(* CoDeSys 2.3.9.62 project: P_auto.pro *)
(* Libraries: Standard.LIB 4.10.05 12:14:46, Iecsfc.lib 2.6.14 11:37:46 *)

(* Global variable list: Global_Variables *)
VAR_GLOBAL
(*Constantes globales*)
	vc:INT:=3; (*Velocidad de las cintas*)
	vagv:INT:=3;
(*Actuadores*)
	GirarIZQ:BOOL;
	Volver1:BOOL;
	Volver2:BOOL;
	GirarA:BOOL;
	GirarB:BOOL;
	GirarC:BOOL;
(*Sensores*)
	Sqr1:INT;
	Sqr2:INT;
	SSC:BOOL;
	SSI:BOOL;
	SSD:BOOL;
	B11:BOOL;
	B12:BOOL;
	B13:BOOL;
	B21:BOOL;
	B22:BOOL;
	B23:BOOL;
	B24: BOOL;
(* Sensores Jorge*)
	sec1:BOOL;
	sec2:BOOL;
	sec3:BOOL;
	sfc1:BOOL;
	sfc2:BOOL;
	sfc3:BOOL;
	sfcint:BOOL;
	ocupado:BOOL;
	secint:BOOL;
(*Almacenes*)
	AlmA:INT:=0;
	AlmB:INT:=0;
	AlmC:INT:=0;
(*AGV*)
	carga1:BOOL;
	carga2:BOOL;
	carga3:BOOL;
(* Camiones*)
	C1:BOOL:=0;
	almc1:INT:=0;
	C2:BOOL:=0;
	almc2:INT:=0;
	C3:BOOL:=0;
	almc3:INT:=0;

(*Visualización de paquetes*)
	pale:ARRAY[0..100] OF paquete;

(* Actuadores cinta principal*)
	disp_paquete:BOOL;
	disp_paquetea:BOOL:=FALSE;
	acp: BOOL; (*Actuador cinta principal*)
	aca: BOOL; (*Actuador cinta A*)
	acb: BOOL; (*Actuador cinta B*)
	acc: BOOL; (*Actuador cinta C*)
	acint:BOOL;(*Actuador cinta intermedia*)
	pasoA:BOOL;(*Paso de cinta A a la intermedia*)
	pasoB:BOOL;(*Paso de cinta B a la intermedia*)
	pasoC:BOOL;(*Paso de cinta C a la intermedia*)
	ac1: BOOL; (*Actuador cinta 1*)
	ac2: BOOL; (*Actuador cinta 2*)
	ac3: BOOL; (*Actuador cinta 3*)
	paq_carga:INT:=0;(*Paquete que esta cargando el brazo*)

(* Sensores cinta principal*)
	scpe: BOOL;
	scps: BOOL;

(* Sensores cintas A, B y C*)
	scae: BOOL;
	scas:BOOL;
	scbe:BOOL;
	scbs:BOOL;
	scce:BOOL;
	sccs:BOOL;

(* Visualización de AGVs *)
	a1:agv;
	a2:agv;
	a3:agv;

(*Rodillo mesa central*)
	rodillo_h_izq: BOOL;
	rodillo_h_drch: BOOL;
	rodillo_v: BOOL;

(* Procesos *)
	spa:BOOL;
	spb:BOOL;
	spc:BOOL;
	cajac1: INT;
	carga: BOOL;
	spgc: BOOL;
	P_ca: BOOL;
	rreset_cca: BOOL;
	reset_cca: BOOL;
	caja_qr: INT;
	Metercola: BOOL;
	P1cola: INT;
	Quitarcola: BOOL;
	reset_ccb: BOOL;
	ld_cb: BOOL;
	reset_cc: BOOL;
	ld_cc: BOOL;
	salidaca: BOOL;
	salidacb: BOOL;
	salidacc: BOOL;
	Quitarcola2: BOOL;
	caja_int: INT;
	P1cola2: INT;
	salidacint: BOOL;
	reset_cint: BOOL;
	ld_cint: BOOL;
	PA: BOOL;
	PB: BOOL;
	PC: BOOL;
	SS3: BOOL;
	SS2: BOOL;
	SS1: BOOL;
	SS0: BOOL;
	sccint: BOOL;
	Girando: BOOL;
	aca1: BOOL;
	aca2: BOOL;
	acb2: BOOL;
	acc2: BOOL;
	salidacc2: BOOL;
	salidacb2: BOOL;
	salidaca2: BOOL;
	reset_contc1: BOOL;
	cajac2: INT;
	cajac3: INT;
	reset_contc2: BOOL;
	reset_contc3: BOOL;
	caja_qr2: INT;
	leer: BOOL;
	pedido: BOOL;
	PedidoTotal: ARRAY[1..3] OF INT;
	c1pais:BOOL;
	c1mundo:BOOL;
	c1abc:BOOL;
	c2pais:BOOL;
	c2mundo:BOOL;
	c2abc:BOOL;
	c3pais:BOOL;
	c3mundo:BOOL;
	c3abc:BOOL;
	descarga: BOOL;
	marcha:BOOL;
	PedidoC1:ARRAY[1..3] OF INT;
	PedidoC2:ARRAY[1..3] OF INT;
	PedidoC3:ARRAY[1..3] OF INT;
	finentrega: BOOL;

	bandera: BOOL;
END_VAR

(* Data type *)
TYPE agv :
STRUCT
	x:INT;
	y:INT;
END_STRUCT
END_TYPE

(* Data type *)
TYPE paquete :
STRUCT
	x:INT;
	y:INT;
	on:BOOL;
	tipo:INT; (*1-->A 2-->B 3-->C*)
	leido:BOOL;
END_STRUCT
END_TYPE

(* POU PLC_PRG, ST *)
PROGRAM PLC_PRG
VAR
END_VAR
Simulador;
vis_cintas;
vis_agv;
Control;
END_PROGRAM

(* POU Visualizacion/Simulador, ST *)
PROGRAM Simulador
VAR
(*Estado*)
	Giro1:INT;
	Giro2:INT;
	Giro3: INT;

END_VAR
(*Actuadores*)
IF Sqr1=1 THEN
GirarIZQ:=1;
END_IF

IF Sqr1=2 THEN
Volver1:=1;
END_IF

IF GirarIZQ=1 THEN
	IF Giro1<>-90 THEN
		Giro1:=Giro1-2;
	END_IF
END_IF;

IF Sqr1=3 THEN
GirarIZQ:=1;
END_IF


IF Sqr2=1 THEN
GirarA:=1;
END_IF

IF GirarA=1 THEN
	IF Giro2 <> -135 THEN
		Giro2:=Giro2-1;
	END_IF
	IF Giro2=-135 THEN
	pale[paq_carga].x:=1230;
	pale[paq_carga].y:=-1300;
	pale[paq_carga].on:=TRUE;
	GirarA:=0;
	END_IF
END_IF;

IF Sqr2=2 THEN
GirarB:=1;
END_IF

IF GirarB=1 THEN
	IF Giro2 <> 180 THEN
		Giro2:=Giro2+1;
	END_IF
	IF Giro2=180 THEN
pale[paq_carga].x:=1450;
	pale[paq_carga].y:=-1230;
	pale[paq_carga].on:=TRUE;
	GirarB:=0;
	END_IF
END_IF;

IF Sqr2=3 THEN
GirarC:=1;
END_IF

IF GirarC=1 THEN
	IF Giro2 <> 135 THEN
		Giro2:=Giro2+1;
	END_IF
	IF Giro2=135 THEN
	pale[paq_carga].x:=1690;
	pale[paq_carga].y:=-1300;
	pale[paq_carga].on:=TRUE;
	GirarC:=0;
      	END_IF
END_IF;

IF Volver1=1 THEN
	IF Giro1<>0 THEN
			Giro1:=Giro1+2;
	END_IF
END_IF;

IF Sqr2=4 THEN
Volver2:=1;
END_IF

IF Volver2=1 THEN
	IF Giro2<>0 THEN
		IF Giro2<0 AND Giro2<>0 THEN
			Giro2:=Giro2+2;
		END_IF;
		IF Giro2>0 AND Giro2<>0  THEN
			Giro2:=Giro2-2;
		END_IF;
	END_IF;
	Volver2:=0;
END_IF;
(*Sensores*)
IF Giro1>=-3 AND Giro1<=3 THEN
	SSC:=1;
ELSE
	SSC:=0;
END_IF

IF Giro1>=-93 AND Giro1<=-87 THEN
	SSI:=1;
ELSE
	SSI:=0;
END_IF


IF Giro2>=135 AND Giro2<=138 THEN
	SS3:=1;
ELSE
	SS3:=0;
END_IF

IF Giro2>=180 AND Giro2<=183 THEN
	SS2:=1;
ELSE
	SS2:=0;
END_IF

IF Giro2>=-138AND Giro2<=-135 THEN
	SS1:=1;
ELSE
	SS1:=0;
END_IF

IF Giro1>=87 AND Giro2<=93 THEN
	SSD:=1;
ELSE
	SSD:=0;
END_IF

IF Giro2>=-3 AND Giro2<=3THEN
	SS0:=1;
ELSE
	SS0:=0;
END_IF


IF B11=1 THEN
	Sqr1:=1;
END_IF

IF B12=1 THEN
	Sqr1:=2;
END_IF

IF B13=1 THEN
	Sqr1:=3;
END_IF

IF B21=1 THEN
	Sqr2:=1;
END_IF

IF B22=1 THEN
	Sqr2:=2;
END_IF

IF B24=1 THEN
	Sqr2:=4;
END_IF


IF B23=1 THEN
	Sqr2:=3;
END_IF
END_PROGRAM

(* POU Visualizacion/vis_cintas, ST *)
PROGRAM vis_cintas (*En esta POU se gestionará todo lo que tenga que ver con la visualización de las cintas. Tanto el funcionamiento de los sensores y actuadores como la gestión de los paquetes que vayan pasando por ellas.*)
VAR
	i: INT:=0; (*Índice que recorre el vector pale, que contiene los paquetes*)
	n:INT:=5; (*Número de paquetes*)
	j:INT:=0;
	ja:INT:=0;
	jb: INT := 0;
	jc:INT:=0;
	jint: INT:=0;
	jbr: INT:=0;
	jalm:INT:=0;
	j1:INT:=0;
	j2:INT:=0;
	j3:INT:=0;
	k:INT:=0;
	ii:INT:=0;
END_VAR
(*Cinta Principal*)

IF disp_paquete AND NOT disp_paquetea	 THEN (*Detector de paquetes por flanco de subida*)
	ii:=ii+1;
	pale[ii].x:=0;
	pale[ii].y:=0;
	pale[ii].on:=TRUE;


	IF ii>=n+1 THEN (*Si hay stack overflow se reinicia el índice*)
		ii:=0;
		bandera:=1;
	END_IF;

END_IF;
disp_paquetea:=disp_paquete;
pale[1].tipo:=1;
pale[2].tipo:=2;
pale[3].tipo:=3;
pale[4].tipo:=3;
pale[5].tipo:=1;


(*Sensor scpe*)
FOR k:=1 TO 5 BY 1 DO
	IF pale[k].y <= 20 AND pale[k].y >=-20 AND pale[k].x >= -20 AND pale[k].x <= 20 AND pale[k].on THEN
		scpe:=TRUE;
		caja_qr:=k;
	EXIT;
	ELSE
	scpe:=FALSE;
	END_IF;

END_FOR

(*Sensor qr*)
FOR k:=1 TO 5 BY 1 DO
	IF pale[k].y <= -271 AND pale[k].y >= -281 AND pale[k].x >= -20 AND pale[k].x <= 20 AND pale[k].on THEN
		leer:=TRUE;
		caja_qr2:=k;
		pale[k].leido:=TRUE;
	EXIT;
	ELSE
	leer:=FALSE;
	END_IF;

END_FOR

(*Sensores Jorge*)
FOR k:=1 TO 5 BY 1 DO
IF pale[k].y <= -1290 AND pale[k].y >=-1330 AND pale[k].x >= 1210AND pale[k].x <= 1250 AND pale[k].on THEN
	sec1:=TRUE;
EXIT;
ELSE
	sec1:=FALSE;
END_IF;END_FOR;
FOR k:=1 TO 5 BY 1 DO
IF pale[k].y <= -1225AND pale[k].y >=-1330 AND pale[k].x >= 1430 AND pale[k].x <=1470AND pale[k].on THEN
	sec2:=TRUE;
EXIT;
ELSE
	sec2:=FALSE;
END_IF;END_FOR;
FOR k:=1 TO 5 BY 1 DO
IF pale[k].y <= -1290 AND pale[k].y >=-1330AND pale[k].x >= 1670  AND pale[k].x <= 1710 AND pale[k].on THEN
	sec3:=TRUE;
EXIT;
ELSE
	sec3:=FALSE;
END_IF;END_FOR;
FOR k:=1 TO 5 BY 1 DO
IF pale[k].y <= -930  AND pale[k].y >=-970 AND pale[k].x >=1040 AND pale[k].x <= 1080 AND pale[k].on THEN
	sfc1:=TRUE;
	cajac1:=k;
EXIT;
ELSE
	sfc1:=FALSE;
END_IF;END_FOR;
FOR k:=1 TO 5 BY 1 DO
IF pale[k].y <= -930AND pale[k].y >=-970 AND pale[k].x >= 1430 AND pale[k].x <=1470AND pale[k].on THEN
	sfc2:=TRUE;
	cajac2:=k;
EXIT;
ELSE
	sfc2:=FALSE;
END_IF;END_FOR;
FOR k:=1 TO 5 BY 1 DO
IF pale[k].y <= -930 AND pale[k].y >=-970 AND pale[k].x >= 1840 AND pale[k].x <= 1880 AND pale[k].on THEN
	sfc3:=TRUE;
	cajac3:=k;
EXIT;
ELSE
	sfc3:=FALSE;
END_IF;END_FOR;
FOR k:=1 TO 5 BY 1 DO
IF pale[k].y <= -1850AND pale[k].y >=-1890 AND pale[k].x >= 1450 AND pale[k].x <=1490AND pale[k].on THEN
	sfcint:=TRUE;
	paq_carga:=k;
EXIT;
ELSE
	sfcint:=FALSE;
END_IF;END_FOR;

FOR k:=1 TO 5 BY 1 DO
IF pale[k].y <= -1850AND pale[k].y >=-1890 AND pale[k].x >= 1400 AND pale[k].x <=1440AND pale[k].on THEN
	sccint:=TRUE;
EXIT;
ELSE
	sccint:=FALSE;
END_IF;END_FOR;

FOR k:=1 TO 5 BY 1 DO
IF pale[k].y <= -1320AND pale[k].y >= -1450AND pale[k].x >= -60AND pale[k].x <=60AND pale[k].on THEN
	ocupado:=TRUE;
	caja_int:=k;
EXIT;
ELSE
	ocupado:=FALSE;
END_IF;END_FOR;
FOR k:=1 TO 5 BY 1 DO
IF pale[k].y <= -1440AND pale[k].y >= -1460AND pale[k].x >= -20AND pale[k].x <=20AND pale[k].on THEN
		secint:=TRUE;
EXIT;
ELSE
	secint:=FALSE;
END_IF;END_FOR;
(*Fin sensores Jorge*)
(*Sensor scps*)
FOR k:=1 TO 5 BY 1 DO
IF pale[k].y >= -490 AND pale[k].y <=-450 AND pale[k].x >= -20 AND pale[k].x <= 20 AND pale[k].on THEN
	scps:=TRUE;
EXIT;
ELSE
	scps:=FALSE;
END_IF;
END_FOR;
(* Sensor scae*)
FOR k:=1 TO 5 BY 1 DO
IF pale[k].x >= -150 AND pale[k].x <=-110 AND pale[k].y >= -630 AND pale[k].y <= -590 AND pale[k].on THEN
	scae:=TRUE;
EXIT;
ELSE
	scae:=FALSE;
END_IF;
END_FOR;
(* Sensor scas*)
FOR k:=1 TO 5 BY 1 DO
IF pale[k].x >= -80 AND pale[k].x <=-60 AND pale[k].y >= -1410 AND pale[k].y <= -1370 AND pale[k].on THEN
	scas:=TRUE;
EXIT;
ELSE
	scas:=FALSE;
END_IF;
END_FOR;
(* Sensor scbe*)
FOR k:=1 TO 5 BY 1 DO
IF pale[k].x >= -20 AND pale[k].x <=20 AND pale[k].y >= -770 AND pale[k].y <= -710 AND pale[k].on THEN
	scbe:=TRUE;
EXIT;
ELSE
	scbe:=FALSE;
END_IF

END_FOR;
(* Sensor scbs*)
FOR k:=1 TO 5 BY 1 DO
IF pale[k].x >= -20 AND pale[k].x <= 20 AND pale[k].y >= -1350 AND pale[k].y <= -1300 AND pale[k].on THEN
	scbs:=TRUE;
EXIT;
ELSE
	scbs:=FALSE;
END_IF;

END_FOR;
(* Sensor scce*)
FOR k:=1 TO 5 BY 1 DO
IF pale[k].x >= 110 AND pale[k].x <= 170 AND pale[k].y >= -630 AND pale[k].y <= -590 AND pale[k].on THEN
	scce:=TRUE;
EXIT;
ELSE
	scce:=FALSE;
END_IF;

END_FOR;
(* Sensor sccs*)
FOR k:=1 TO 5 BY 1 DO
IF pale[k].x >= 50 AND pale[k].x <= 90 AND pale[k].y >= -1410 AND pale[k].y <= -1370 AND pale[k].on THEN
	sccs:=TRUE;
EXIT;
ELSE
	sccs:=FALSE;
END_IF;
END_FOR;
(*Actuador acp*)
IF acp THEN
	FOR j:=1 TO 5 DO
	IF pale[j].y >= -610AND pale[j].y <=0  AND pale[j].on THEN
		pale[j].y:=pale[j].y-vc;

	END_IF;
	END_FOR;
END_IF;
(*Actuador aca*)

IF aca THEN
	FOR ja:=1 TO 5 DO
	IF pale[ja].x >= -423 AND pale[ja].x <=-100 AND pale[ja].y >= -630 AND pale[ja].y <= -590 AND pale[ja].on THEN
		pale[ja].x:=pale[ja].x-vc;

	END_IF;
	IF pale[ja].x >= -427 AND pale[ja].x <=-423 THEN
		IF pale[ja].y >= -1055 AND pale[ja].y <=-605 THEN
		 pale[ja].y:=pale[ja].y-vc;
		END_IF;
	END_IF;
	END_FOR;
END_IF;
IF aca2 THEN
	FOR ja:=1 TO 5 DO
		IF pale[ja].x >= -427 AND pale[ja].x <=-423 THEN
			IF pale[ja].y >= -1393 AND pale[ja].y <=-1055THEN
		 	pale[ja].y:=pale[ja].y-vc;
			END_IF;
		END_IF;
		IF pale[ja].y >= -1395 AND pale[ja].y <=-1390 THEN
			IF pale[ja].x >= -427 AND pale[ja].x <=0THEN
			pale[ja].x:=pale[ja].x+vc;
			END_IF;

		END_IF;
END_FOR;
END_IF;
(*Actuador acc*)
IF acc THEN
	FOR jc:=1 TO 5 DO
	IF pale[jc].y >= -612 AND pale[jc].y <=-605 THEN
		IF pale[jc].x >= 100 AND pale[jc].x <=425 THEN
		pale[jc].x:=pale[jc].x+vc;
		END_IF;
	END_IF;
	IF pale[jc].x >= 423 AND pale[jc].x <=427THEN
		IF pale[jc].y >= -1055 AND pale[jc].y <=-605 THEN
		 pale[jc].y:=pale[jc].y-vc;
		END_IF;
	END_IF;
	END_FOR;
END_IF;
IF acc2 THEN
	FOR jc:=1 TO 5 DO
	IF pale[jc].x >= 423 AND pale[jc].x <=427THEN
		IF pale[jc].y >= -1393 AND pale[jc].y <=-1055 THEN
		 pale[jc].y:=pale[jc].y-vc;
		END_IF;
	END_IF;
	IF pale[jc].y >= -1395 AND pale[jc].y <=-1390 THEN
		IF pale[jc].x >= 0 AND pale[jc].x <=425THEN
		pale[jc].x:=pale[jc].x-vc;
		END_IF;

	END_IF;
	END_FOR;
END_IF;
(*Actuador acb*)
IF acb THEN
	FOR jb:=1 TO 5 DO
		IF pale[jb].x>=-3 AND pale[jb].x <= 3 THEN
		IF pale[jb].y >= -1055AND pale[jb].y <=-730 THEN
		 pale[jb].y:=pale[jb].y-vc;
		END_IF
		END_IF;
	END_FOR;
END_IF;

IF acb2 THEN
	FOR jb:=1 TO 5 DO
		IF pale[jb].x>=-3 AND pale[jb].x <= 3 THEN
		IF pale[jb].y >= -1395 AND pale[jb].y <=-1055 THEN
		 pale[jb].y:=pale[jb].y-vc;
		END_IF
		END_IF;
	END_FOR;
END_IF;
(*Rodillos*)
IF rodillo_h_izq THEN
	FOR i:=1 TO 5 DO
		IF pale[i].x>= -110 AND pale[i].x<= 3 AND pale[i].y >= -630 AND pale[i].y <= -590 AND pale[i].on THEN
		   pale[i].x:=pale[i].x-vc;
		END_IF
	END_FOR
END_IF


IF rodillo_h_drch THEN
	FOR i:=1 TO 5 DO
		IF pale[i].x>= -3 AND pale[i].x<=110 AND pale[i].y >= -630 AND pale[i].y <= -590 AND pale[i].on THEN
		   pale[i].x:=pale[i].x+vc;
		END_IF
	END_FOR
END_IF

IF rodillo_v THEN
	FOR i:=1 TO 5 DO
		IF pale[i].x>=-3 AND pale[i].x<=3 AND pale[i].y >= -730 AND pale[i].y <= -590 AND pale[i].on THEN
			pale[i].y:=pale[i].y-vc;
		END_IF
	END_FOR
END_IF


(*Actuador acint*)
IF acint THEN
	FOR jint:=1 TO 5 DO
	IF pale[jint].x>=-3 AND pale[jint].x<=3 THEN
		IF pale[jint].y >= -1880 AND pale[jint].y <= -1365 THEN
		pale[jint].y:=pale[jint].y-vc;
		END_IF
	END_IF
	IF pale[jint].y>=-1883 AND pale[jint].y<=-1877 THEN
		IF pale[jint].x>=-3 AND pale[jint].x<=1460 THEN
		pale[jint].x:=pale[jint].x + vc;
		END_IF
	END_IF
	END_FOR
END_IF
(*Actuador ac1*)
IF ac1 THEN
	FOR j1:=1 TO 5 DO
	IF pale[j1].x>=1227AND pale[j1].x<=1233 THEN
		IF pale[j1].y >= -1303AND pale[j1].y <= -950THEN
		pale[j1].y:=pale[j1].y+vc;
		END_IF
	END_IF
	IF pale[j1].y>=-953 AND pale[j1].y<=-947THEN
		IF pale[j1].x>=1060 AND pale[j1].x<=1230 THEN
		pale[j1].x:=pale[j1].x - vc;
		END_IF
	END_IF
	END_FOR
END_IF
(*Actuador ac2*)
IF ac2 THEN
	FOR j2:=1 TO 5 DO
	IF pale[j2].x>=1447AND pale[j2].x<=1453 THEN
		IF pale[j2].y >= -1303AND pale[j2].y <= -950THEN
		pale[j2].y:=pale[j2].y+vc;
		END_IF
	END_IF
	END_FOR
END_IF
(*Actuador ac3*)
IF ac3 THEN
	FOR j3:=1 TO 5 DO
	IF pale[j3].x>=1687AND pale[j3].x<=1693 THEN
		IF pale[j3].y >= -1303AND pale[j3].y <= -950 THEN
		pale[j3].y:=pale[j3].y+vc;
		END_IF
	END_IF
	IF pale[j3].y>=-953 AND pale[j3].y<=-947 THEN
		IF pale[j3].x>=1687 AND pale[j3].x<=1860 THEN
		pale[j3].x:=pale[j3].x + vc;
		END_IF
	END_IF
	END_FOR
END_IF

(*Brazo robótico*)
IF GirarA OR GirarB OR GirarC THEN
	pale[paq_carga].on:=FALSE;
END_IF
(*
FOR jbr:=1 TO 5 DO
	IF pale[jbr].x>=1457 AND pale[jbr].x<=1463 THEN
		IF pale[jbr].y>=-1883 AND pale[jbr].y<=1877 THEN

				paq_carga:=jbr;
				pale[paq_carga].on:=FALSE;
			END_IF
			IF GirarB=1 AND pale[jbr].tipo=2 THEN
				paq_carga:=jbr;
				pale[paq_carga].on:=FALSE;
			END_IF
			IF GirarC=1 AND pale[jbr].tipo=3 THEN
				paq_carga:=jbr;
				pale[paq_carga].on:=FALSE;
			END_IF
		END_IF
	END_IF
END_FOR

(*Almacen*)

FOR jalm:=1 TO 5 DO
	IF pale[jalm].y>=-953 AND pale[jalm].y<=-947 THEN
		IF pale[jalm].x>=1057AND pale[jalm].x<=1063THEN
			AlmA:=AlmA+1;
			pale[jalm].on:=FALSE;
			pale[jalm].x:=0;
			pale[jalm].y:=0;
		END_IF
		IF pale[jalm].x>=1447 AND pale[jalm].x<=1453 THEN
			AlmB:=AlmB+1;
			pale[jalm].on:=FALSE;
			pale[jalm].x:=0;
			pale[jalm].y:=0;
		END_IF
		IF pale[jalm].x>=1857 AND pale[jalm].x<=1863 THEN
			AlmC:=AlmC+1;
			pale[jalm].on:=FALSE;
			pale[jalm].x:=0;
			pale[jalm].y:=0;
		END_IF
	END_IF
END_FOR
*)
(* Procesos *)
(*C*)
FOR i:=1 TO 5 BY 1 DO
IF pale[i].x >= 400 AND pale[i].x <= 440 AND pale[i].y >= -1060 AND pale[i].y <= -1020 THEN
spc:=TRUE;
EXIT;
ELSE
spc:=FALSE;
END_IF;
END_FOR;

(*B*)
FOR i:=1 TO 5 BY 1 DO
	IF pale[i].x >= -20 AND pale[i].x <= 20 AND pale[i].y >= -1060 AND pale[i].y <= -1020 AND pale[i].on THEN
		spb:=TRUE;
		EXIT;
	ELSE
		spb:=FALSE;
	END_IF;
END_FOR;

(*A*)
FOR i:=1 TO 5 BY 1 DO
IF pale[i].x >= -440 AND pale[i].x <= -400 AND pale[i].y >= -1060 AND pale[i].y <= -1020 THEN
spa:=TRUE;
EXIT;
ELSE
spa:=FALSE;
END_IF;
END_FOR;
(*plataforma giratoria*)
FOR i:=1 TO 5 BY 1 DO
IF pale[i].x >= -20 AND pale[i].x <= 20 AND pale[i].y >= -632 AND pale[i].y <= -592 AND pale[i].on THEN
spgc:=TRUE;
EXIT;
ELSE
spgc:=FALSE;
END_IF;
END_FOR;
END_PROGRAM

(* POU Visualizacion/vis_agv, ST *)
PROGRAM vis_agv
VAR

END_VAR
IF marcha THEN
	IF a1.x >=-15 AND a1.x <= 5 AND a1.y >= -10 AND a1.y <= 615 THEN
	a1.y:=a1.y+vagv;

	ELSIF a1.x <= 5 AND a1.x >= -765 AND a1.y <= 620 AND a1.y >= 610 THEN
	a1.x:=a1.x-vagv;

	ELSIF a1.x >= -770 AND a1.x <=-760 AND a1.y <= 620 AND a1.y >= -5 THEN
	a1.y:=a1.y-vagv;

	ELSIF a1.x >= -770 AND a1.x <=10 AND a1.y <= 10 AND a1.y >= -10 THEN
	a1.x:=a1.x+vagv;
	END_IF;

END_IF;

IF marcha THEN


	IF a2.x >= -10 AND a2.x <=770 AND a2.y <= 10 AND a2.y >= -10 THEN
	a2.x:=a2.x+vagv;

	ELSIF a2.x >=760 AND a2.x <= 780 AND a2.y >= -10 AND a2.y <= 615 THEN
	a2.y:=a2.y+vagv;

	ELSIF a2.x <= 780 AND a2.x >= -5 AND a2.y <= 620 AND a2.y >= 610 THEN
	a2.x:=a2.x-vagv;

	ELSIF a2.x >= -10 AND a2.x <=10 AND a2.y <= 620 AND a2.y >= -5 THEN
	a2.y:=a2.y-vagv;


	END_IF;

END_IF;


IF marcha THEN


	IF a3.x >= -10 AND a3.x <=395 AND a3.y <= 10 AND a3.y >= -10 THEN
	a3.x:=a3.x+vagv;

	ELSIF a3.x >=390 AND a3.x <= 400 AND a3.y >= -10 AND a3.y <= 615 THEN
	a3.y:=a3.y+vagv;

	ELSIF a3.x <= 400 AND a3.x >= -370 AND a3.y <= 620 AND a3.y >= 610 THEN
	a3.x:=a3.x-vagv;

	ELSIF a3.x >= -375 AND a3.x <=-365 AND a3.y <= 620 AND a3.y >= -5 THEN
	a3.y:=a3.y-vagv;

	ELSIF a3.x >= -375 AND a3.x <=5 AND a3.y <= 10 AND a3.y >= -10 THEN
	a3.x:=a3.x+vagv;

	END_IF;

END_IF;

(*Sensores de carga*)

(* Sensor 1*)

IF a1.x >= -20 AND  a1.x <= 20 AND a1.y >= -20 AND a1.y <= 20 THEN

carga3:=TRUE;

ELSE

carga3:=FALSE;

END_IF;

(*Sensor 2*)
IF a2.x >= -20 AND  a2.x <= 20 AND a2.y >= -20 AND a2.y <= 20 THEN


carga2:=TRUE;

ELSE

carga2:=FALSE;

END_IF;

(*Sensor 3*)
IF a3.x >= -20 AND  a3.x <= 20 AND a3.y >= -20 AND a3.y <= 20 THEN


carga1:=TRUE;

ELSE

carga1:=FALSE;

END_IF;

(*Sensores de descarga*)

(* Sensor 1*)

IF a1.x >= -20 AND  a1.x <= 20 AND a1.y >= 590 AND a1.y <= 630 OR  a2.x >= 740 AND  a2.x <= 780 AND a2.y >= 590 AND a2.y <= 630 OR a3.x >= 370 AND  a3.x <= 440 AND a3.y >= 590 AND a3.y <= 630  THEN

C1:=TRUE;

ELSE

C1:=FALSE;

END_IF;

(* Sensor 2*)

IF a1.x >= -410 AND  a1.x <= -370 AND a1.y >= 590 AND a1.y <= 630 OR  a2.x >= 350 AND  a2.x <= 390 AND a2.y >= 590 AND a2.y <= 630 OR a3.x >= -20 AND  a3.x <= 20 AND a3.y >= 590 AND a3.y <= 630  THEN

C2:=TRUE;

ELSE

C2:=FALSE;

END_IF;

(* Sensor 3*)

IF a1.x >= -780 AND  a1.x <= -740 AND a1.y >= 590 AND a1.y <= 630 OR  a2.x >= -20 AND  a2.x <= 20 AND a2.y >= 590 AND a2.y <= 630 OR a3.x >= -390 AND  a3.x <= -350 AND a3.y >= 590 AND a3.y <= 630  THEN

C3:=TRUE;

ELSE

C3:=FALSE;

END_IF;
END_PROGRAM

(* POU Modos/Control, SFC *)
PROGRAM Control
VAR
END_VAR
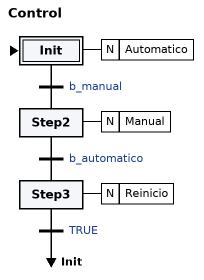
INITIAL_STEP Init:
	Automatico(N);
END_STEP
TRANSITION FROM Init TO Step2 := b_manual;
END_TRANSITION
STEP Step2:
	Manual(N);
END_STEP
TRANSITION FROM Step2 TO Step3 := b_automatico;
END_TRANSITION
STEP Step3:
	Reinicio(N);
END_STEP
TRANSITION FROM Step3 TO Init := TRUE;
END_TRANSITION
END_PROGRAM

(* POU Modos/Automatico, ST *)
PROGRAM Automatico
VAR
END_VAR
cp;
pg;
lectorqr;
cintas123;
CintaINT;
AUX;
Brazo;
CintasABC;
almacen;
camiones;
AGV_AUX;
AGVS;
Dispensador;
END_PROGRAM

(* POU Auto/cp, SFC *)
PROGRAM cp
VAR
END_VAR
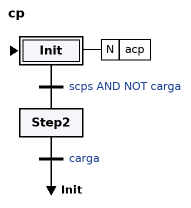
INITIAL_STEP Init:
	acp(N);
END_STEP
TRANSITION FROM Init TO Step2 := scps AND NOT carga;
END_TRANSITION
STEP Step2:
END_STEP
TRANSITION FROM Step2 TO Init := carga;
END_TRANSITION
END_PROGRAM

(* POU Auto/pg, SFC *)
PROGRAM pg
VAR
	u: INT;
	Trans0: BOOL;
	Trans5: BOOL;
	Trans7: BOOL;
	Trans3: BOOL;
	scbe_trig: F_TRIG;
	scae_trig: F_TRIG;
	scce_trig: F_TRIG;
END_VAR
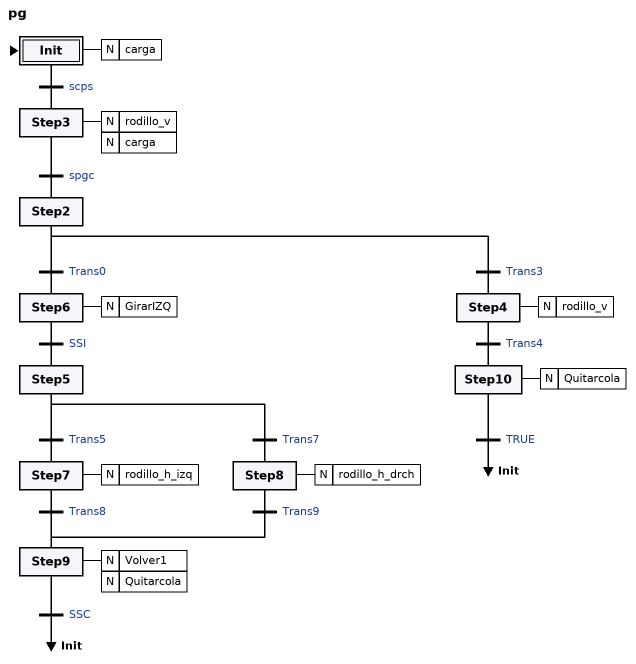
INITIAL_STEP Init:
	carga(N);
END_STEP
TRANSITION FROM Init TO Step3 := scps;
END_TRANSITION
STEP Step3:
	rodillo_v(N);
	carga(N);
END_STEP
TRANSITION FROM Step3 TO Step2 := spgc;
END_TRANSITION
STEP Step2:
END_STEP
TRANSITION FROM Step2 TO Step6 := Trans0;
END_TRANSITION
TRANSITION FROM Step2 TO Step4 := Trans3;
END_TRANSITION
STEP Step6:
	GirarIZQ(N);
END_STEP
TRANSITION FROM Step6 TO Step5 := SSI;
END_TRANSITION
STEP Step5:
END_STEP
TRANSITION FROM Step5 TO Step7 := Trans5;
END_TRANSITION
TRANSITION FROM Step5 TO Step8 := Trans7;
END_TRANSITION
STEP Step7:
	rodillo_h_izq(N);
END_STEP
TRANSITION FROM Step7 TO Step9 := Trans8;
END_TRANSITION
STEP Step8:
	rodillo_h_drch(N);
END_STEP
TRANSITION FROM Step8 TO Step9 := Trans9;
END_TRANSITION
STEP Step9:
	Volver1(N);
	Quitarcola(N);
END_STEP
TRANSITION FROM Step9 TO Init := SSC;
END_TRANSITION
STEP Step4:
	rodillo_v(N);
END_STEP
TRANSITION FROM Step4 TO Step10 := Trans4;
END_TRANSITION
STEP Step10:
	Quitarcola(N);
END_STEP
TRANSITION FROM Step10 TO Init := TRUE;
END_TRANSITION

TRANSITION Trans0:
 P1cola<>2
END_TRANSITION

TRANSITION Trans5:
P1cola=1
END_TRANSITION

TRANSITION Trans8:
_LD_ (* Ladder Diagram *)
NETWORK 1
	[scae] - scae_trig:F_TRIG(CLK: *)
_END_LD_
(* the same logic as Structured Text *)
(* Network 1 *)
scae_trig(CLK := scae);
Trans8 := scae_trig.Q;
END_TRANSITION

TRANSITION Trans7:
	 P1cola=3
END_TRANSITION

TRANSITION Trans9:
_LD_ (* Ladder Diagram *)
NETWORK 1
	[scce] - scce_trig:F_TRIG(CLK: *)
_END_LD_
(* the same logic as Structured Text *)
(* Network 1 *)
scce_trig(CLK := scce);
Trans9 := scce_trig.Q;
END_TRANSITION

TRANSITION Trans3:
P1cola=2
END_TRANSITION

TRANSITION Trans4:
_LD_ (* Ladder Diagram *)
NETWORK 1
	[scbe] - scbe_trig:F_TRIG(CLK: *)
_END_LD_
(* the same logic as Structured Text *)
(* Network 1 *)
scbe_trig(CLK := scbe);
Trans4 := scbe_trig.Q;
END_TRANSITION
END_PROGRAM

(* POU Auto/lectorqr, ST *)
PROGRAM lectorqr

VAR
	cola: ARRAY[0..12] OF INT;
	Metercolaa:BOOL;
	Quitarcolaa:BOOL;
	N:INT;
	I:INT;
END_VAR
IF scpe=1 AND Metercolaa=0 THEN
	cola[N]:=pale[caja_qr].tipo;
	N:=N+1;
END_IF

Metercolaa:=scpe;
P1cola:=cola[0];
IF Quitarcola=1 AND Quitarcolaa=0 THEN
	FOR i:=0 TO N-1 BY 1 DO
		cola[i]:=cola[i+1];
	END_FOR
	N:=N-1;
END_IF
Quitarcolaa:=Quitarcola;
END_PROGRAM

(* POU Auto/cintas123, LD *)
PROGRAM cintas123
VAR
	contc1: CTUD;
	P_c1: BOOL;
	contc2: CTUD;
	P_c2: BOOL;
	contc3: CTUD;
	P_c3: BOOL;
END_VAR
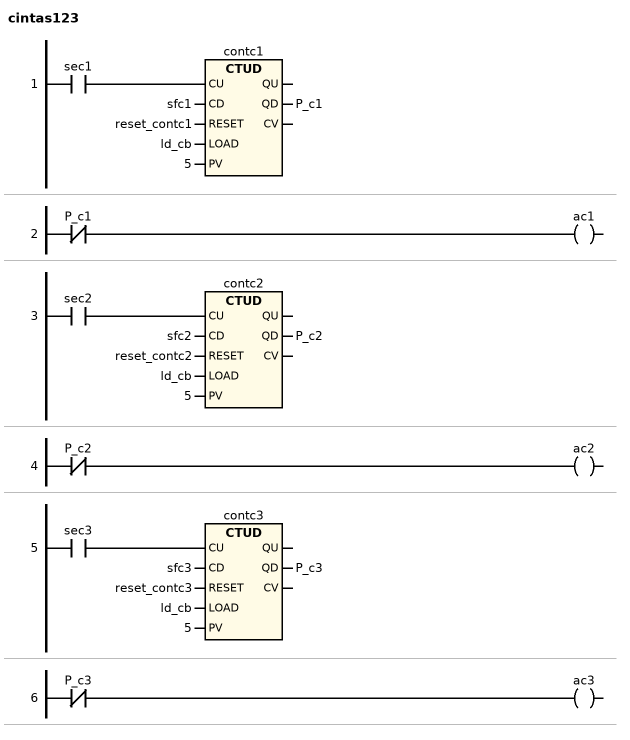
_LD_ (* Ladder Diagram *)
NETWORK 1
	[sec1] - contc1:CTUD(CU: *, CD: sfc1, RESET: reset_contc1, LOAD: ld_cb, PV: 5, QD => P_c1)
NETWORK 2
	[/P_c1] --- (ac1)
NETWORK 3
	[sec2] - contc2:CTUD(CU: *, CD: sfc2, RESET: reset_contc2, LOAD: ld_cb, PV: 5, QD => P_c2)
NETWORK 4
	[/P_c2] --- (ac2)
NETWORK 5
	[sec3] - contc3:CTUD(CU: *, CD: sfc3, RESET: reset_contc3, LOAD: ld_cb, PV: 5, QD => P_c3)
NETWORK 6
	[/P_c3] --- (ac3)
_END_LD_
(* the same logic as Structured Text *)
(* Network 1 *)
contc1(CU := sec1, CD := sfc1, RESET := reset_contc1, LOAD := ld_cb, PV := 5);
P_c1 := contc1.QD;
(* Network 2 *)
ac1 := NOT P_c1;
(* Network 3 *)
contc2(CU := sec2, CD := sfc2, RESET := reset_contc2, LOAD := ld_cb, PV := 5);
P_c2 := contc2.QD;
(* Network 4 *)
ac2 := NOT P_c2;
(* Network 5 *)
contc3(CU := sec3, CD := sfc3, RESET := reset_contc3, LOAD := ld_cb, PV := 5);
P_c3 := contc3.QD;
(* Network 6 *)
ac3 := NOT P_c3;
END_PROGRAM

(* POU Auto/CintaINT, LD *)
PROGRAM CintaINT
VAR
	Timer1: TON;
	EncenderCint: BOOL;
	P_cint: BOOL;
	COUNTER_CINT: CTUD;
END_VAR
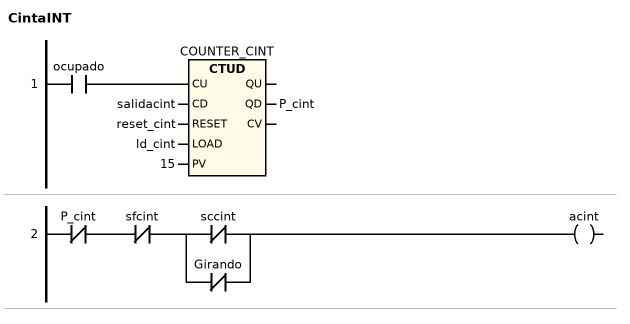
_LD_ (* Ladder Diagram *)
NETWORK 1
	[ocupado] - COUNTER_CINT:CTUD(CU: *, CD: salidacint, RESET: reset_cint, LOAD: ld_cint, PV: 15, QD => P_cint)
NETWORK 2
	[/P_cint] - [/sfcint] - { [/sccint] | [/Girando] } --- (acint)
_END_LD_
(* the same logic as Structured Text *)
(* Network 1 *)
COUNTER_CINT(CU := ocupado, CD := salidacint, RESET := reset_cint, LOAD := ld_cint, PV := 15);
P_cint := COUNTER_CINT.QD;
(* Network 2 *)
acint := NOT P_cint AND NOT sfcint AND (NOT sccint OR NOT Girando);
END_PROGRAM

(* POU Auto/AUX, ST *)
PROGRAM AUX
VAR
	scasa: BOOL;
	scbsa: BOOL;
	sccsa: BOOL;
	Metercolaa: BOOL;
	N: INT;
	Quitarcolaa: BOOL;
	i: INT;
	cola2:ARRAY[0..12] OF INT;
	sfcinta: BOOL;
	spca: BOOL;
	spba: BOOL;
	spaa: BOOL;
END_VAR
IF sfcint=0 AND sfcinta=1 THEN
	salidacint:=1;
ELSE
	salidacint:=0;
END_IF
sfcinta:=sfcint;


IF ocupado=1 AND Metercolaa=0 THEN
	cola2[N]:=pale[caja_int].tipo;
	N:=N+1;
END_IF

Metercolaa:=ocupado;
P1cola2:=cola2[0];
IF Quitarcola2=1 AND Quitarcolaa=0 THEN
	FOR i:=0 TO N-1 BY 1 DO
		cola2[i]:=cola2[i+1];
	END_FOR
	N:=N-1;
END_IF
Quitarcolaa:=Quitarcola2;
END_PROGRAM

(* POU Auto/Brazo, SFC *)
PROGRAM Brazo
VAR
END_VAR
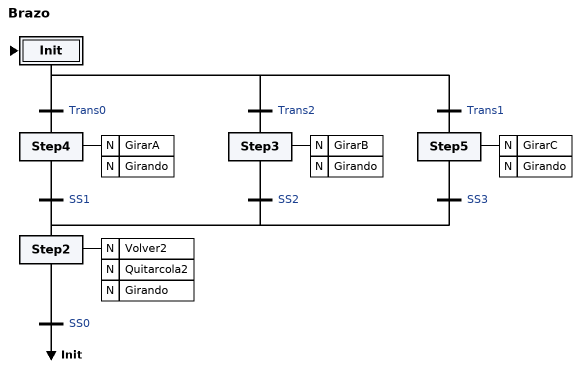
INITIAL_STEP Init:
END_STEP
TRANSITION FROM Init TO Step4 := Trans0;
END_TRANSITION
TRANSITION FROM Init TO Step3 := Trans2;
END_TRANSITION
TRANSITION FROM Init TO Step5 := Trans1;
END_TRANSITION
STEP Step4:
	GirarA(N);
	Girando(N);
END_STEP
TRANSITION FROM Step4 TO Step2 := SS1;
END_TRANSITION
STEP Step3:
	GirarB(N);
	Girando(N);
END_STEP
TRANSITION FROM Step3 TO Step2 := SS2;
END_TRANSITION
STEP Step5:
	GirarC(N);
	Girando(N);
END_STEP
TRANSITION FROM Step5 TO Step2 := SS3;
END_TRANSITION
STEP Step2:
	Volver2(N);
	Quitarcola2(N);
	Girando(N);
END_STEP
TRANSITION FROM Step2 TO Init := SS0;
END_TRANSITION

TRANSITION Trans0:
sfcint=1 AND P1cola2=1
END_TRANSITION

TRANSITION Trans2:
sfcint=1 AND P1cola2=2
END_TRANSITION

TRANSITION Trans1:
sfcint=1 AND P1cola2=3
END_TRANSITION
END_PROGRAM

(* POU Auto/CintasABC, LD *)
PROGRAM CintasABC
VAR
	COUNTER_CA: CTUD;
	ld_ca: BOOL;
	COUNTER_CB: CTUD;
	P_cb: BOOL;
	COUNTER_CC: CTUD;
	P_cc: BOOL;
	ocupado_trig: F_TRIG;
	Timer1: TON;
	salidaca2s: BOOL;
	salidacb2s: BOOL;
	Timer2: TON;
	Timer3: TON;
	salidacc2s: BOOL;
	spa_trigger: R_TRIG;
	T_Encartado: TON;
	spb_trigger: R_TRIG;
	spc_trigger: R_TRIG;
	T_Flejado: TON;
	T_Embolsado: TON;
	P_ca2: BOOL;
	salidacc22s: BOOL;
	salidacb22s: BOOL;
	salidaca22s: BOOL;
	COUNTER_CC2: CTUD;
	COUNTER_CB2: CTUD;
	COUNTER_CA2: CTUD;
	P_cb2: BOOL;
	P_cc2: BOOL;
	Timer32: TON;
	Timer22: TON;
	Timer12: TON;
	spc_trigger2: F_TRIG;
	spc_trigger3: F_TRIG;
	spa_trigger2: F_TRIG;
	spa_trigger3: F_TRIG;
	salidaa: BOOL;
	salidab: BOOL;
	spb_trigger3: F_TRIG;
	salidac: BOOL;
	spb_trigger2: F_TRIG;
END_VAR
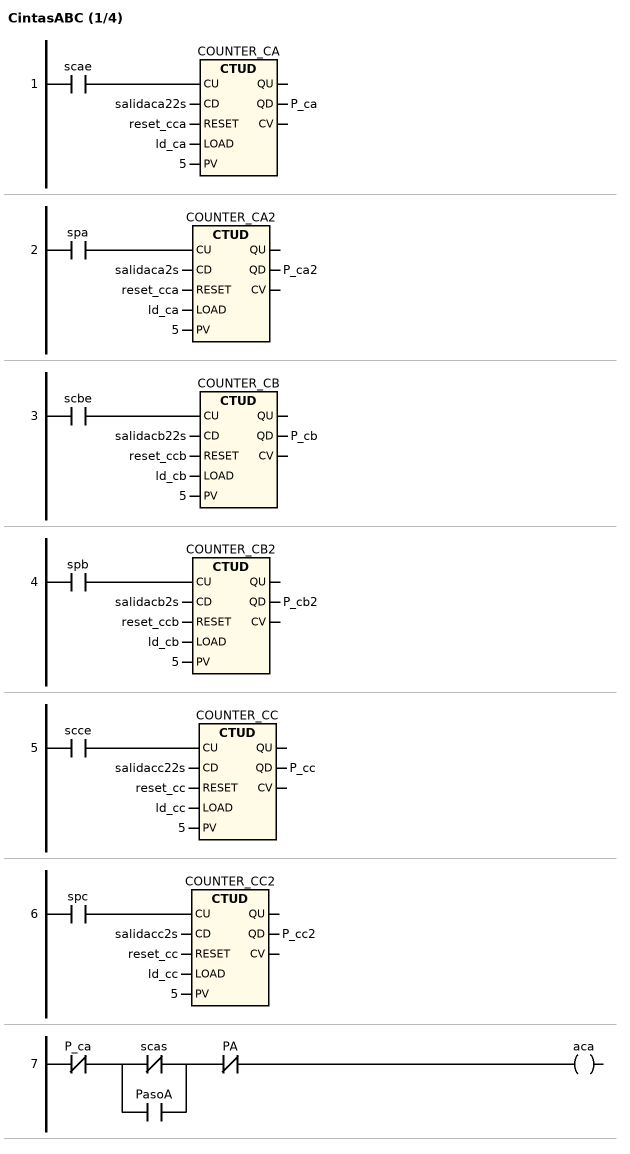
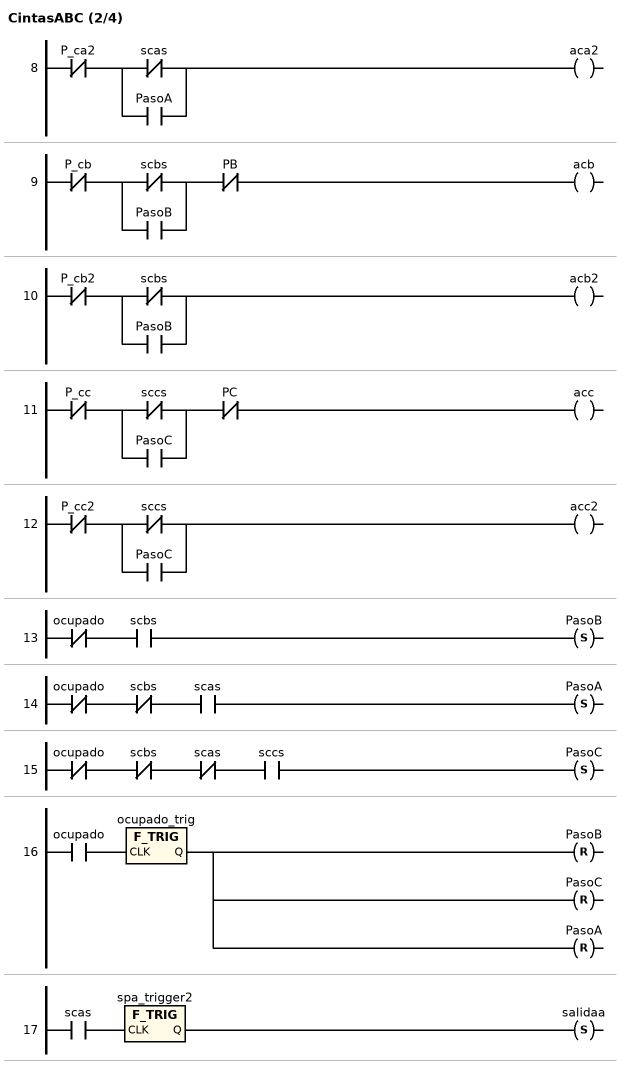
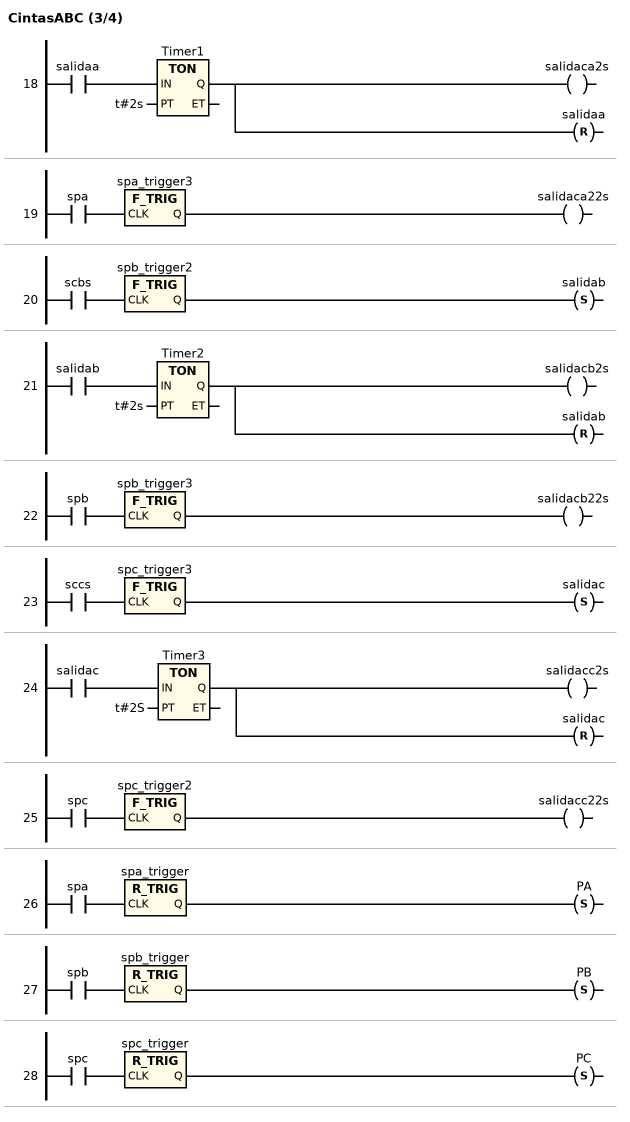
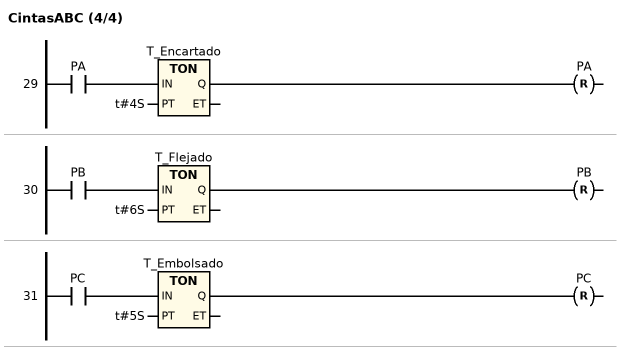
_LD_ (* Ladder Diagram *)
NETWORK 1
	[scae] - COUNTER_CA:CTUD(CU: *, CD: salidaca22s, RESET: reset_cca, LOAD: ld_ca, PV: 5, QD => P_ca)
NETWORK 2
	[spa] - COUNTER_CA2:CTUD(CU: *, CD: salidaca2s, RESET: reset_cca, LOAD: ld_ca, PV: 5, QD => P_ca2)
NETWORK 3
	[scbe] - COUNTER_CB:CTUD(CU: *, CD: salidacb22s, RESET: reset_ccb, LOAD: ld_cb, PV: 5, QD => P_cb)
NETWORK 4
	[spb] - COUNTER_CB2:CTUD(CU: *, CD: salidacb2s, RESET: reset_ccb, LOAD: ld_cb, PV: 5, QD => P_cb2)
NETWORK 5
	[scce] - COUNTER_CC:CTUD(CU: *, CD: salidacc22s, RESET: reset_cc, LOAD: ld_cc, PV: 5, QD => P_cc)
NETWORK 6
	[spc] - COUNTER_CC2:CTUD(CU: *, CD: salidacc2s, RESET: reset_cc, LOAD: ld_cc, PV: 5, QD => P_cc2)
NETWORK 7
	[/P_ca] - { [/scas] | [PasoA] } - [/PA] --- (aca)
NETWORK 8
	[/P_ca2] - { [/scas] | [PasoA] } --- (aca2)
NETWORK 9
	[/P_cb] - { [/scbs] | [PasoB] } - [/PB] --- (acb)
NETWORK 10
	[/P_cb2] - { [/scbs] | [PasoB] } --- (acb2)
NETWORK 11
	[/P_cc] - { [/sccs] | [PasoC] } - [/PC] --- (acc)
NETWORK 12
	[/P_cc2] - { [/sccs] | [PasoC] } --- (acc2)
NETWORK 13
	[/ocupado] - [scbs] --- (S PasoB)
NETWORK 14
	[/ocupado] - [/scbs] - [scas] --- (S PasoA)
NETWORK 15
	[/ocupado] - [/scbs] - [/scas] - [sccs] --- (S PasoC)
NETWORK 16
	[ocupado] - ocupado_trig:F_TRIG(CLK: *) --- (R PasoB) (R PasoC) (R PasoA)
NETWORK 17
	[scas] - spa_trigger2:F_TRIG(CLK: *) --- (S salidaa)
NETWORK 18
	[salidaa] - Timer1:TON(IN: *, PT: t#2s) --- (salidaca2s) (R salidaa)
NETWORK 19
	[spa] - spa_trigger3:F_TRIG(CLK: *) --- (salidaca22s)
NETWORK 20
	[scbs] - spb_trigger2:F_TRIG(CLK: *) --- (S salidab)
NETWORK 21
	[salidab] - Timer2:TON(IN: *, PT: t#2s) --- (salidacb2s) (R salidab)
NETWORK 22
	[spb] - spb_trigger3:F_TRIG(CLK: *) --- (salidacb22s)
NETWORK 23
	[sccs] - spc_trigger3:F_TRIG(CLK: *) --- (S salidac)
NETWORK 24
	[salidac] - Timer3:TON(IN: *, PT: t#2S) --- (salidacc2s) (R salidac)
NETWORK 25
	[spc] - spc_trigger2:F_TRIG(CLK: *) --- (salidacc22s)
NETWORK 26
	[spa] - spa_trigger:R_TRIG(CLK: *) --- (S PA)
NETWORK 27
	[spb] - spb_trigger:R_TRIG(CLK: *) --- (S PB)
NETWORK 28
	[spc] - spc_trigger:R_TRIG(CLK: *) --- (S PC)
NETWORK 29
	[PA] - T_Encartado:TON(IN: *, PT: t#4S) --- (R PA)
NETWORK 30
	[PB] - T_Flejado:TON(IN: *, PT: t#6S) --- (R PB)
NETWORK 31
	[PC] - T_Embolsado:TON(IN: *, PT: t#5S) --- (R PC)
_END_LD_
(* the same logic as Structured Text *)
(* Network 1 *)
COUNTER_CA(CU := scae, CD := salidaca22s, RESET := reset_cca, LOAD := ld_ca, PV := 5);
P_ca := COUNTER_CA.QD;
(* Network 2 *)
COUNTER_CA2(CU := spa, CD := salidaca2s, RESET := reset_cca, LOAD := ld_ca, PV := 5);
P_ca2 := COUNTER_CA2.QD;
(* Network 3 *)
COUNTER_CB(CU := scbe, CD := salidacb22s, RESET := reset_ccb, LOAD := ld_cb, PV := 5);
P_cb := COUNTER_CB.QD;
(* Network 4 *)
COUNTER_CB2(CU := spb, CD := salidacb2s, RESET := reset_ccb, LOAD := ld_cb, PV := 5);
P_cb2 := COUNTER_CB2.QD;
(* Network 5 *)
COUNTER_CC(CU := scce, CD := salidacc22s, RESET := reset_cc, LOAD := ld_cc, PV := 5);
P_cc := COUNTER_CC.QD;
(* Network 6 *)
COUNTER_CC2(CU := spc, CD := salidacc2s, RESET := reset_cc, LOAD := ld_cc, PV := 5);
P_cc2 := COUNTER_CC2.QD;
(* Network 7 *)
aca := NOT P_ca AND (NOT scas OR PasoA) AND NOT PA;
(* Network 8 *)
aca2 := NOT P_ca2 AND (NOT scas OR PasoA);
(* Network 9 *)
acb := NOT P_cb AND (NOT scbs OR PasoB) AND NOT PB;
(* Network 10 *)
acb2 := NOT P_cb2 AND (NOT scbs OR PasoB);
(* Network 11 *)
acc := NOT P_cc AND (NOT sccs OR PasoC) AND NOT PC;
(* Network 12 *)
acc2 := NOT P_cc2 AND (NOT sccs OR PasoC);
(* Network 13 *)
IF NOT ocupado AND scbs THEN PasoB := TRUE; END_IF;
(* Network 14 *)
IF NOT ocupado AND NOT scbs AND scas THEN PasoA := TRUE; END_IF;
(* Network 15 *)
IF NOT ocupado AND NOT scbs AND NOT scas AND sccs THEN PasoC := TRUE; END_IF;
(* Network 16 *)
ocupado_trig(CLK := ocupado);
IF ocupado_trig.Q THEN PasoB := FALSE; PasoC := FALSE; PasoA := FALSE; END_IF;
(* Network 17 *)
spa_trigger2(CLK := scas);
IF spa_trigger2.Q THEN salidaa := TRUE; END_IF;
(* Network 18 *)
Timer1(IN := salidaa, PT := t#2s);
salidaca2s := Timer1.Q;
IF Timer1.Q THEN salidaa := FALSE; END_IF;
(* Network 19 *)
spa_trigger3(CLK := spa);
salidaca22s := spa_trigger3.Q;
(* Network 20 *)
spb_trigger2(CLK := scbs);
IF spb_trigger2.Q THEN salidab := TRUE; END_IF;
(* Network 21 *)
Timer2(IN := salidab, PT := t#2s);
salidacb2s := Timer2.Q;
IF Timer2.Q THEN salidab := FALSE; END_IF;
(* Network 22 *)
spb_trigger3(CLK := spb);
salidacb22s := spb_trigger3.Q;
(* Network 23 *)
spc_trigger3(CLK := sccs);
IF spc_trigger3.Q THEN salidac := TRUE; END_IF;
(* Network 24 *)
Timer3(IN := salidac, PT := t#2S);
salidacc2s := Timer3.Q;
IF Timer3.Q THEN salidac := FALSE; END_IF;
(* Network 25 *)
spc_trigger2(CLK := spc);
salidacc22s := spc_trigger2.Q;
(* Network 26 *)
spa_trigger(CLK := spa);
IF spa_trigger.Q THEN PA := TRUE; END_IF;
(* Network 27 *)
spb_trigger(CLK := spb);
IF spb_trigger.Q THEN PB := TRUE; END_IF;
(* Network 28 *)
spc_trigger(CLK := spc);
IF spc_trigger.Q THEN PC := TRUE; END_IF;
(* Network 29 *)
T_Encartado(IN := PA, PT := t#4S);
IF T_Encartado.Q THEN PA := FALSE; END_IF;
(* Network 30 *)
T_Flejado(IN := PB, PT := t#6S);
IF T_Flejado.Q THEN PB := FALSE; END_IF;
(* Network 31 *)
T_Embolsado(IN := PC, PT := t#5S);
IF T_Embolsado.Q THEN PC := FALSE; END_IF;
END_PROGRAM

(* POU Auto/almacen, ST *)
PROGRAM almacen
VAR
END_VAR
IF sfc1=1 THEN
	pale[cajac1].x:=0;
	pale[cajac1].y:=0;
	pale[cajac1].leido:=FALSE;
	pale[cajac1].on:=FALSE;
	AlmA:=AlmA+1;
END_IF

IF sfc2=1 THEN
	pale[cajac2].x:=0;
	pale[cajac2].y:=0;
	pale[cajac2].leido:=FALSE;
	pale[cajac2].on:=FALSE;
	AlmB:=AlmB+1;
END_IF

IF sfc3=1 THEN
	pale[cajac3].x:=0;
	pale[cajac3].y:=0;
	pale[cajac3].leido:=FALSE;
	pale[cajac3].on:=FALSE;
	AlmC:=AlmC+1;
END_IF
END_PROGRAM

(* POU Auto/camiones, ST *)
PROGRAM camiones
VAR
	c1paisa:BOOL;
	c1abca:BOOL;
	c1mundoa:BOOL;
	c2paisa:BOOL;
	c2abca:BOOL;
	c2mundoa:BOOL;
	c3paisa:BOOL;
	c3abca:BOOL;
	c3mundoa:BOOL;
END_VAR
IF c1pais=1 AND c1paisa=0 THEN
	PedidoC1[1]:=PedidoC1[1]+1;
END_IF
c1paisa:=c1pais;
IF c1abc=1 AND c1abca=0 THEN
	PedidoC1[2]:=PedidoC1[2]+1;
END_IF
c1abca:=c1abc;
IF c1mundo=1 AND c1mundoa=0 THEN
	PedidoC1[3]:=PedidoC1[3]+1;
END_IF
c1mundoa:=c1mundo;
IF c2pais=1 AND c2paisa=0 THEN
	PedidoC2[1]:=PedidoC2[1]+1;
END_IF
c2paisa:=c2pais;
IF c2abc=1 AND c2abca=0 THEN
	PedidoC2[2]:=PedidoC2[2]+1;
END_IF
c2abca:=c2abc;
IF c2mundo=1 AND c2mundoa=0 THEN
	PedidoC2[3]:=PedidoC2[3]+1;
END_IF
c2mundoa:=c2mundo;
IF c3pais=1 AND c3paisa=0 THEN
	PedidoC3[1]:=PedidoC3[1]+1;
END_IF
c3paisa:=c3pais;
IF c3abc=1 AND c3abca=0 THEN
	PedidoC3[2]:=PedidoC3[2]+1;
END_IF
c3abca:=c3abc;
IF c3mundo=1 AND c3mundoa=0 THEN
	PedidoC3[3]:=PedidoC3[3]+1;
END_IF
c3mundoa:=c3mundo;
IF pedido=1 THEN
	PedidoTotal[1]:=PedidoC1[1]+PedidoC2[1]+PedidoC3[1];
	PedidoTotal[2]:=PedidoC1[2]+PedidoC2[2]+PedidoC3[2];
	PedidoTotal[3]:=PedidoC1[3]+PedidoC2[3]+PedidoC3[3];
END_IF
END_PROGRAM

(* POU Auto/AGV_AUX, ST *)
PROGRAM AGV_AUX
VAR
END_VAR
IF c3=0 AND c2=0 AND c1=1 THEN
	IF PedidoC1[3]<>0 THEN
		descarga:=1;
		PedidoC1[3]:=0;
	END_IF
END_IF

IF c3=0 AND c2=1 AND c1=1 THEN
	IF PedidoC1[2]<>0  OR PedidoC2[3]<>0 THEN
		descarga:=1;
		PedidoC1[2]:=0;
		PedidoC2[3]:=0;
	END_IF
END_IF


IF c3=1 AND c2=1 AND c1=1 THEN
	IF PedidoC1[1]<>0  OR PedidoC2[2]<>0 OR PedidoC1[1]<>0THEN
		descarga:=1;
		PedidoC1[1]:=0;
		PedidoC2[2]:=0;
		PedidoC3[3]:=0;
	END_IF
END_IF


IF c3=1 AND c2=1 AND c1=0 THEN
	IF PedidoC3[2]<>0  OR PedidoC2[1]<>0 THEN
		descarga:=1;
		PedidoC3[2]:=0;
		PedidoC2[1]:=0;
	END_IF
END_IF

IF c3=1 AND c2=0 AND c1=0 THEN
	IF PedidoC3[1]<>0 THEN
		descarga:=1;
		PedidoC3[1]:=0;
		finentrega:=1;
	END_IF
END_IF

IF carga1=1 AND carga2=1 AND carga3=1 AND finentrega=1 THEN
	a1.x:=0;
a1.y:=0;
a2.x:=0;
 a2.y:=0;
a3.x:=0;
a3.y:=0;
	finentrega:=0;
pedido:=0;
END_IF

IF pedido=1 THEN
 IF AlmA<PedidoTotal[1] OR AlmB<PedidoTotal[2] OR AlmC<PedidoTotal[3] THEN
	carga:=1;
ELSE
	carga:=0;
END_IF;
END_IF;
END_PROGRAM

(* POU Auto/AGVS, LD *)
PROGRAM AGVS
VAR
	timer1: TON;
END_VAR
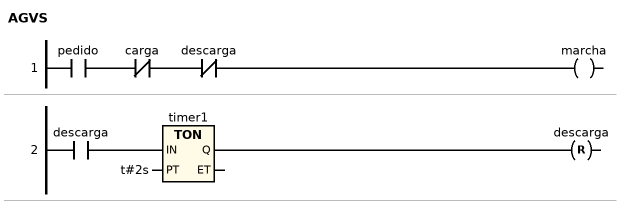
_LD_ (* Ladder Diagram *)
NETWORK 1
	[pedido] - [/carga] - [/descarga] --- (marcha)
NETWORK 2
	[descarga] - timer1:TON(IN: *, PT: t#2s) --- (R descarga)
_END_LD_
(* the same logic as Structured Text *)
(* Network 1 *)
marcha := pedido AND NOT carga AND NOT descarga;
(* Network 2 *)
timer1(IN := descarga, PT := t#2s);
IF timer1.Q THEN descarga := FALSE; END_IF;
END_PROGRAM

(* POU Auto/Dispensador, LD *)
PROGRAM Dispensador
VAR
	timer1: TON;
	soltar_paquete: BOOL;
	trigger: R_TRIG;
END_VAR
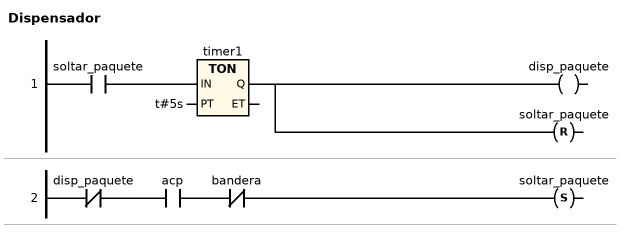
_LD_ (* Ladder Diagram *)
NETWORK 1
	[soltar_paquete] - timer1:TON(IN: *, PT: t#5s) --- (disp_paquete) (R soltar_paquete)
NETWORK 2
	[/disp_paquete] - [acp] - [/bandera] --- (S soltar_paquete)
_END_LD_
(* the same logic as Structured Text *)
(* Network 1 *)
timer1(IN := soltar_paquete, PT := t#5s);
disp_paquete := timer1.Q;
IF timer1.Q THEN soltar_paquete := FALSE; END_IF;
(* Network 2 *)
IF NOT disp_paquete AND acp AND NOT bandera THEN soltar_paquete := TRUE; END_IF;
END_PROGRAM

(* POU Modos/Manual, LD *)
PROGRAM Manual
VAR
	b_paquete: BOOL;
	b_acp: BOOL;
	b_rod_carga: BOOL;
	b_rod_desc: BOOL;
	b_aca: BOOL;
	b_acb: BOOL;
	b_acc: BOOL;
	b_acint: BOOL;
	b_GirarIZQ: BOOL;
	b_Volver1: BOOL;
	b_B21: BOOL;
	b_B22: BOOL;
	b_B23: BOOL;
	b_B24: BOOL;
	b_ac1: BOOL;
	b_ac2: BOOL;
	b_ac3: BOOL;
	b_vis_agv: BOOL;
	b_c1pais: BOOL;
	b_c1abc: BOOL;
	b_c1mundo: BOOL;
	b_c2pais: BOOL;
	b_c2abc: BOOL;
	b_c2mundo: BOOL;
	b_c3pais: BOOL;
	b_c3abc: BOOL;
	b_c3mundo: BOOL;
	b_pedido: BOOL;
END_VAR
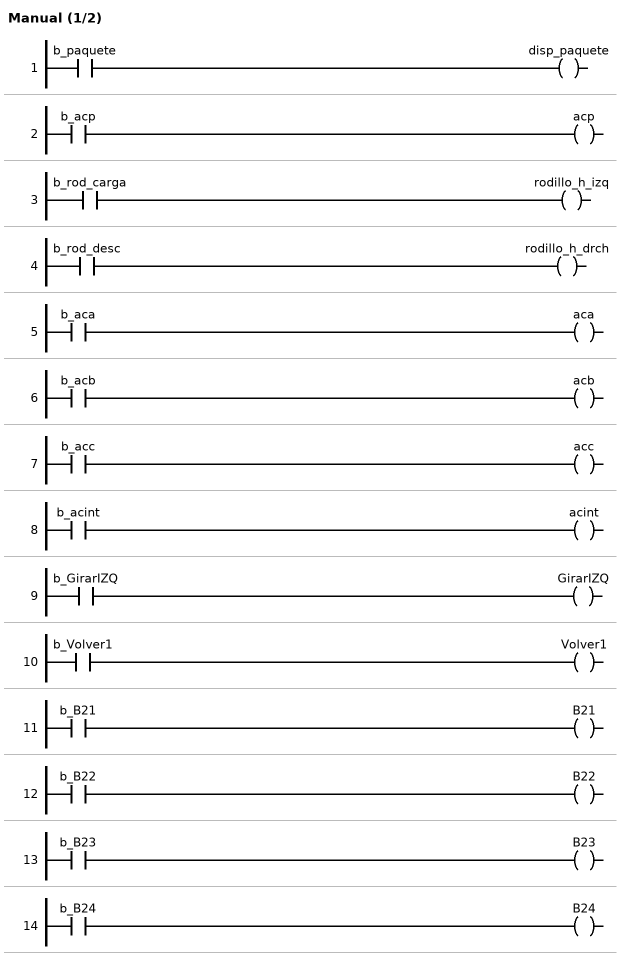
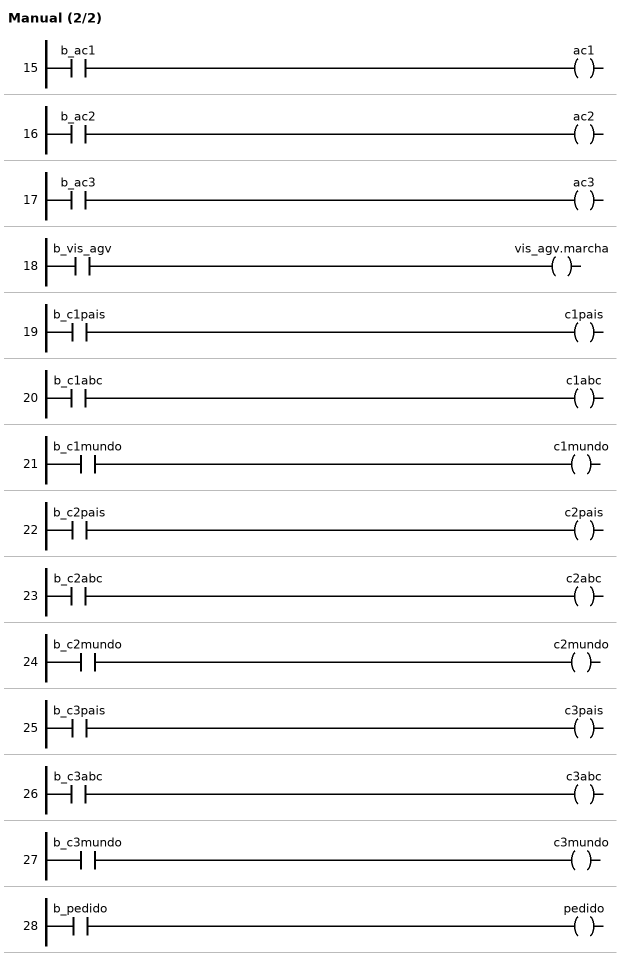
_LD_ (* Ladder Diagram *)
NETWORK 1
	[b_paquete] --- (disp_paquete)
NETWORK 2
	[b_acp] --- (acp)
NETWORK 3
	[b_rod_carga] --- (rodillo_h_izq)
NETWORK 4
	[b_rod_desc] --- (rodillo_h_drch)
NETWORK 5
	[b_aca] --- (aca)
NETWORK 6
	[b_acb] --- (acb)
NETWORK 7
	[b_acc] --- (acc)
NETWORK 8
	[b_acint] --- (acint)
NETWORK 9
	[b_GirarIZQ] --- (GirarIZQ)
NETWORK 10
	[b_Volver1] --- (Volver1)
NETWORK 11
	[b_B21] --- (B21)
NETWORK 12
	[b_B22] --- (B22)
NETWORK 13
	[b_B23] --- (B23)
NETWORK 14
	[b_B24] --- (B24)
NETWORK 15
	[b_ac1] --- (ac1)
NETWORK 16
	[b_ac2] --- (ac2)
NETWORK 17
	[b_ac3] --- (ac3)
NETWORK 18
	[b_vis_agv] --- (vis_agv.marcha)
NETWORK 19
	[b_c1pais] --- (c1pais)
NETWORK 20
	[b_c1abc] --- (c1abc)
NETWORK 21
	[b_c1mundo] --- (c1mundo)
NETWORK 22
	[b_c2pais] --- (c2pais)
NETWORK 23
	[b_c2abc] --- (c2abc)
NETWORK 24
	[b_c2mundo] --- (c2mundo)
NETWORK 25
	[b_c3pais] --- (c3pais)
NETWORK 26
	[b_c3abc] --- (c3abc)
NETWORK 27
	[b_c3mundo] --- (c3mundo)
NETWORK 28
	[b_pedido] --- (pedido)
_END_LD_
(* the same logic as Structured Text *)
(* Network 1 *)
disp_paquete := b_paquete;
(* Network 2 *)
acp := b_acp;
(* Network 3 *)
rodillo_h_izq := b_rod_carga;
(* Network 4 *)
rodillo_h_drch := b_rod_desc;
(* Network 5 *)
aca := b_aca;
(* Network 6 *)
acb := b_acb;
(* Network 7 *)
acc := b_acc;
(* Network 8 *)
acint := b_acint;
(* Network 9 *)
GirarIZQ := b_GirarIZQ;
(* Network 10 *)
Volver1 := b_Volver1;
(* Network 11 *)
B21 := b_B21;
(* Network 12 *)
B22 := b_B22;
(* Network 13 *)
B23 := b_B23;
(* Network 14 *)
B24 := b_B24;
(* Network 15 *)
ac1 := b_ac1;
(* Network 16 *)
ac2 := b_ac2;
(* Network 17 *)
ac3 := b_ac3;
(* Network 18 *)
vis_agv.marcha := b_vis_agv;
(* Network 19 *)
c1pais := b_c1pais;
(* Network 20 *)
c1abc := b_c1abc;
(* Network 21 *)
c1mundo := b_c1mundo;
(* Network 22 *)
c2pais := b_c2pais;
(* Network 23 *)
c2abc := b_c2abc;
(* Network 24 *)
c2mundo := b_c2mundo;
(* Network 25 *)
c3pais := b_c3pais;
(* Network 26 *)
c3abc := b_c3abc;
(* Network 27 *)
c3mundo := b_c3mundo;
(* Network 28 *)
pedido := b_pedido;
END_PROGRAM

(* Visualisation Almacen
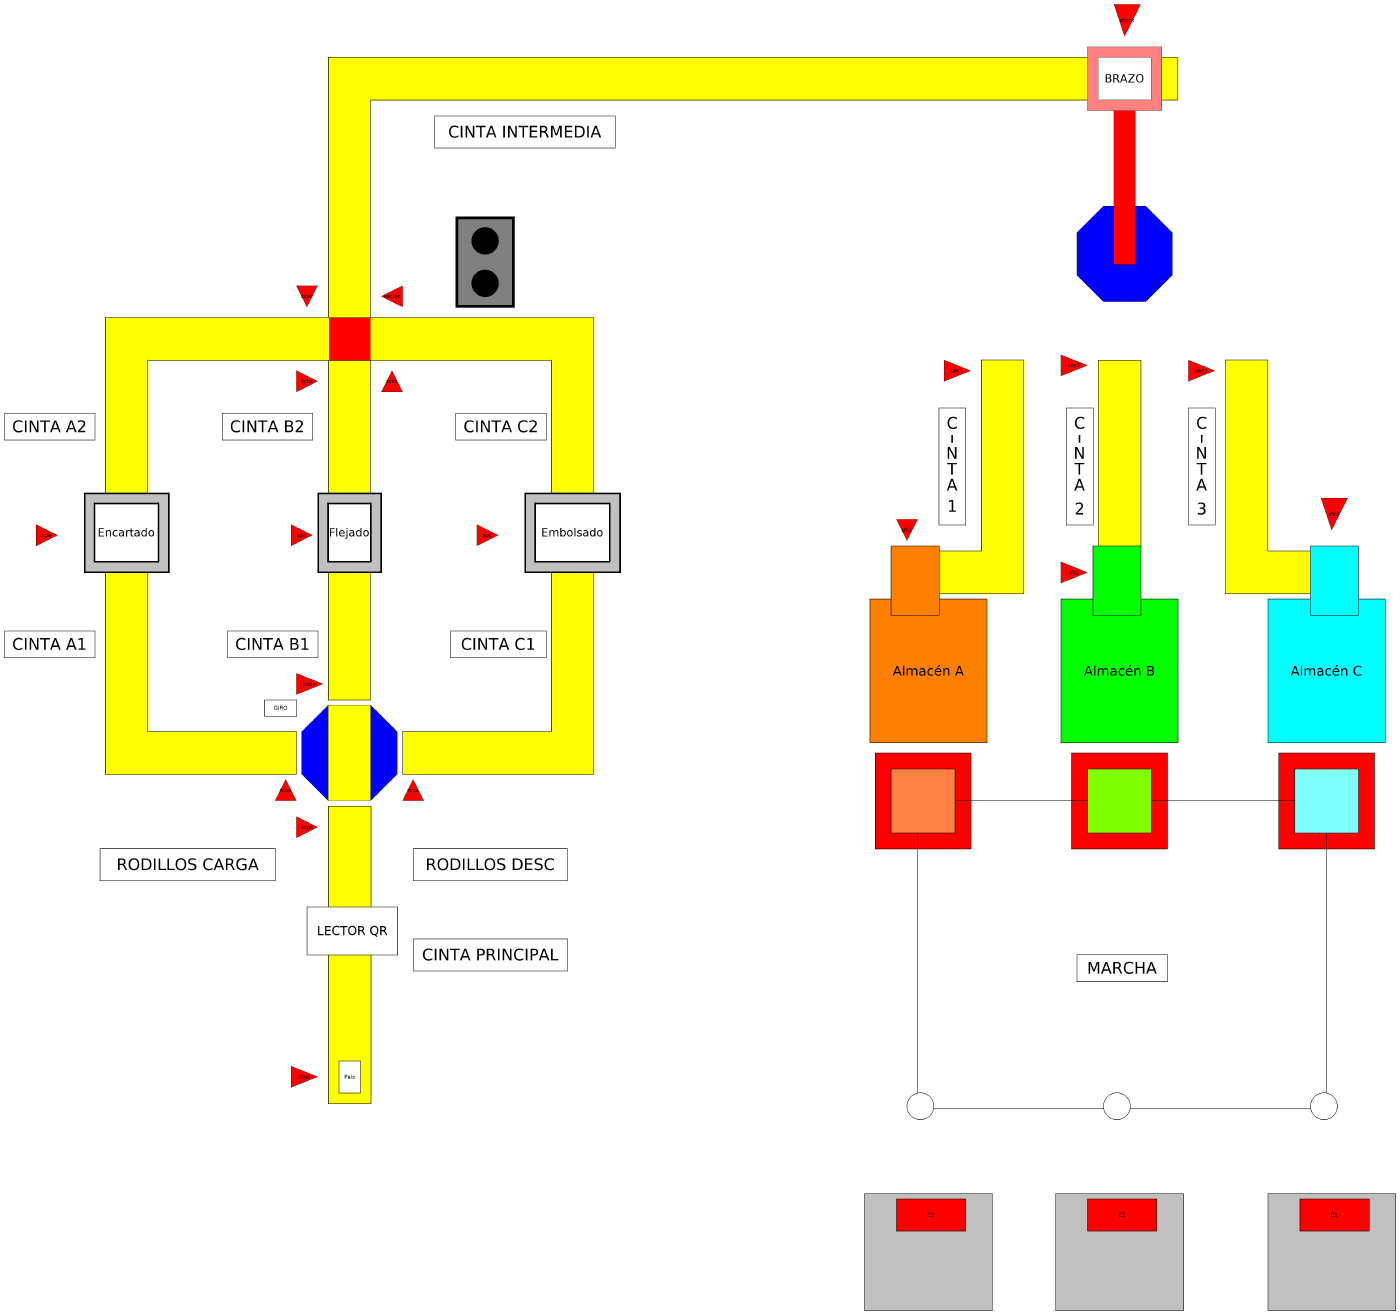
polygon at (2410,830)-(2460,870): text "sec3"; alarm colour if sec3
polygon at (2170,820)-(2220,860): text "sec2"; alarm colour if sec2
polygon at (1950,830)-(2000,870): text "sec1"; alarm colour if sec1
rectangle at (2180,920)-(2231,1141): alarm colour if ac2
rectangle at (2190,1090)-(2221,1131): text "2"; alarm colour if ac2
rectangle at (2190,1050)-(2221,1081): text "A"; alarm colour if ac2
rectangle at (2190,1020)-(2221,1051): text "T"; alarm colour if ac2
rectangle at (2190,990)-(2221,1021): text "N"; alarm colour if ac2
rectangle at (2190,960)-(2221,991): text "I"; alarm colour if ac2
rectangle at (2190,930)-(2221,971): text "C"; alarm colour if ac2
rectangle at (2410,920)-(2461,1141): alarm colour if ac3
rectangle at (2420,1090)-(2451,1131): text "3"; alarm colour if ac3
rectangle at (2420,1050)-(2451,1081): text "A"; alarm colour if ac3
rectangle at (2420,1020)-(2451,1051): text "T"; alarm colour if ac3
rectangle at (2420,990)-(2451,1021): text "N"; alarm colour if ac3
rectangle at (2420,960)-(2451,991): text "I"; alarm colour if ac3
rectangle at (2420,930)-(2451,971): text "C"; alarm colour if ac3
rectangle at (1940,920)-(1991,1141): alarm colour if ac1
rectangle at (2580,1570)-(2761,1751): alarm colour if carga3
rectangle at (2190,1570)-(2371,1751): alarm colour if carga2
rectangle at (1820,1570)-(2001,1751): alarm colour if carga1
rectangle at (790,750)-(871,831): alarm colour if ocupado
rounded rectangle at (1810,1280)-(2031,1551): text "Almacén A"
rounded rectangle at (2170,1280)-(2391,1551): text "Almacén B"
rounded rectangle at (2560,1280)-(2781,1551): text "Almacén C"
polygon at (740,1480)-(920,1660): angle Simulador.Giro1
polygon at (790,1480)-(870,1660): angle Simulador.Giro1
polygon at (2270,300)-(2310,650): angle Simulador.Giro2
rectangle at (810,2150)-(851,2211): text "Pais"; invisible if NOT pale[1].on; alarm colour if pale[1].leido; left pale[1].x; top pale[1].y; right pale[1].x; bottom pale[1].y
polygon at (720,2160)-(770,2200): text "scpe"; alarm colour if scpe
rectangle at (810,2150)-(851,2211): text "ABC"; invisible if NOT pale[2].on; alarm colour if pale[2].leido; left pale[2].x; top pale[2].y; right pale[2].x; bottom pale[2].y
rectangle at (810,2150)-(851,2211): text "Mundo"; invisible if NOT pale[3].on; alarm colour if pale[3].leido; left pale[3].x; top pale[3].y; right pale[3].x; bottom pale[3].y
rectangle at (810,2150)-(851,2211): text "Mundo"; invisible if NOT pale[4].on; alarm colour if pale[4].leido; left pale[4].x; top pale[4].y; right pale[4].x; bottom pale[4].y
rectangle at (810,2150)-(851,2211): text "Pais"; invisible if NOT pale[5].on; alarm colour if pale[5].leido; left pale[5].x; top pale[5].y; right pale[5].x; bottom pale[5].y
polygon at (2220,240)-(2360,360): angle Simulador.Giro2
rectangle at (2610,1600)-(2731,1721): x offset a1.x; y offset a1.y
rectangle at (2220,1600)-(2341,1721): x offset a3.x; y offset a3.y
rectangle at (1850,1600)-(1971,1721): x offset a2.x; y offset a2.y
polygon at (730,1690)-(770,1730): text "scps"; alarm colour if scps
rectangle at (670,1470)-(731,1501): text "GIRO"; alarm colour if SSI
polygon at (690,1620)-(730,1660): text "scae"; alarm colour if scae
polygon at (930,1620)-(970,1660): text "scce"; alarm colour if scce
polygon at (730,1420)-(780,1460): text "scbe"; alarm colour if scbe
polygon at (730,850)-(770,890): text "scbs"; alarm colour if scbs
polygon at (730,690)-(770,730): text "scas"; alarm colour if scas
polygon at (890,850)-(930,890): text "sccs"; alarm colour if sccs
polygon at (890,690)-(930,730): text "secint"; alarm colour if secint
polygon at (2270,160)-(2320,220): text "sfcint"; alarm colour if sfcint
polygon at (2170,1210)-(2220,1250): text "sfc2"; alarm colour if sfc2
polygon at (1860,1130)-(1900,1170): text "sfc1"; alarm colour if sfc1
polygon at (2660,1090)-(2710,1150): text "sfc3"; alarm colour if sfc3
rectangle at (2620,2410)-(2751,2471): text "C3"; alarm colour if c1
rectangle at (2220,2410)-(2351,2471): text "C2"; alarm colour if c2
rectangle at (1860,2410)-(1991,2471): text "C3"; alarm colour if c3
rectangle at (950,1920)-(1241,1981): text "CINTA PRINCIPAL"; alarm colour if acp
rectangle at (180,1340)-(351,1391): text "CINTA A1"; alarm colour if aca
rectangle at (600,1340)-(771,1391): text "CINTA B1"; alarm colour if acb
rectangle at (1020,1340)-(1201,1391): text "CINTA C1"; alarm colour if acc
rectangle at (360,1750)-(691,1811): text "RODILLOS CARGA"; alarm colour if rodillo_h_izq or rodillo_v
rectangle at (950,1750)-(1241,1811): text "RODILLOS DESC"; alarm colour if rodillo_h_drch
ellipse at (1060,580)-(1111,631): alarm colour if ocupado
ellipse at (1060,660)-(1111,711): alarm colour if not(ocupado)
rectangle at (990,370)-(1331,431): text "CINTA INTERMEDIA"; alarm colour if acint
rectangle at (1950,1020)-(1981,1051): text "T"; alarm colour if ac1
rectangle at (1950,1050)-(1981,1081): text "A"; alarm colour if ac1
rectangle at (1950,990)-(1981,1021): text "N"; alarm colour if ac1
rectangle at (1950,1090)-(1981,1121): text "1"; alarm colour if ac1
rectangle at (1950,960)-(1981,991): text "I"; alarm colour if ac1
rectangle at (1950,930)-(1981,971): text "C"; alarm colour if ac1
rectangle at (2200,1950)-(2371,2001): text "MARCHA"; alarm colour if vis_agv.marcha
polygon at (2240,260)-(2340,340): text "BRAZO"; alarm colour if GirarA OR GirarB OR GirarC OR Volver2; angle Simulador.Giro2
polygon at (720,1140)-(760,1180): text "spb"; alarm colour if spb
polygon at (790,1100)-(870,1210): text "Flejado"; alarm colour if PB
polygon at (1070,1140)-(1110,1180): text "spc"; alarm colour if spc
polygon at (1180,1100)-(1320,1210): text "Embolsado"; alarm colour if PC
polygon at (240,1140)-(280,1180): text "spa"; alarm colour if spa
polygon at (350,1100)-(470,1210): text "Encartado"; alarm colour if PA
rectangle at (180,930)-(351,981): text "CINTA A2"; alarm colour if aca2
rectangle at (590,930)-(761,981): text "CINTA B2"; alarm colour if acb2
rectangle at (1030,930)-(1201,981): text "CINTA C2"; alarm colour if acc2
rectangle at (750,1860)-(921,1951): text "LECTOR QR"; alarm colour if leer
36 more shapes without text or variables
*)

(* Visualisation Botonera_alm_agv
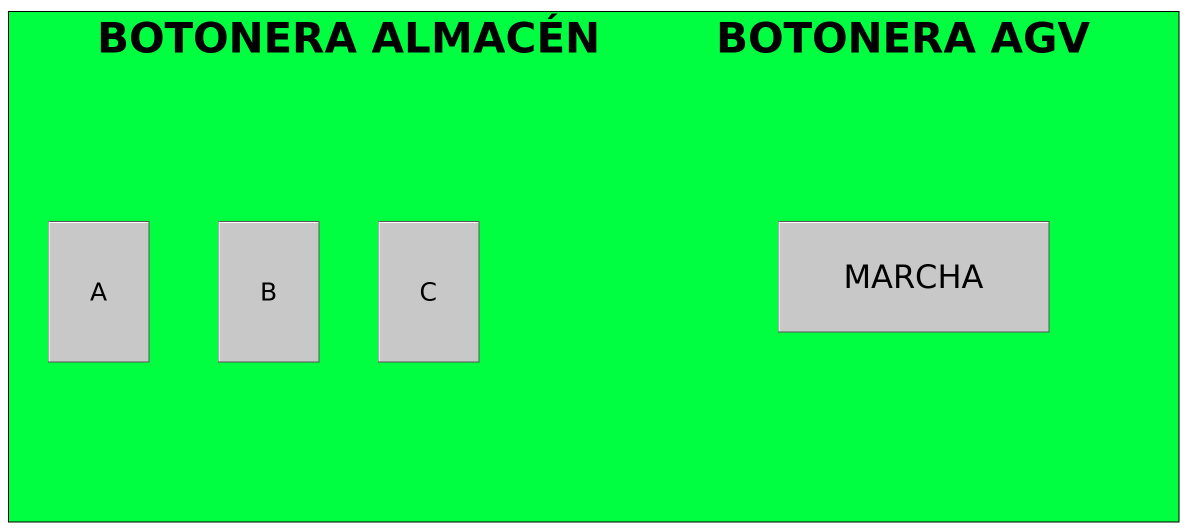
rectangle at (60,60)-(1231,571): text "BOTONERA ALMACÉN        BOTONERA AGV"
button at (100,270)-(201,411): text "A"; toggles b_ac1
button at (270,270)-(371,411): text "B"; toggles b_ac2
button at (430,270)-(531,411): text "C"; toggles b_ac3
button at (830,270)-(1101,381): text "MARCHA"; toggles b_vis_agv
*)

(* Visualisation Botonera_cin_gru
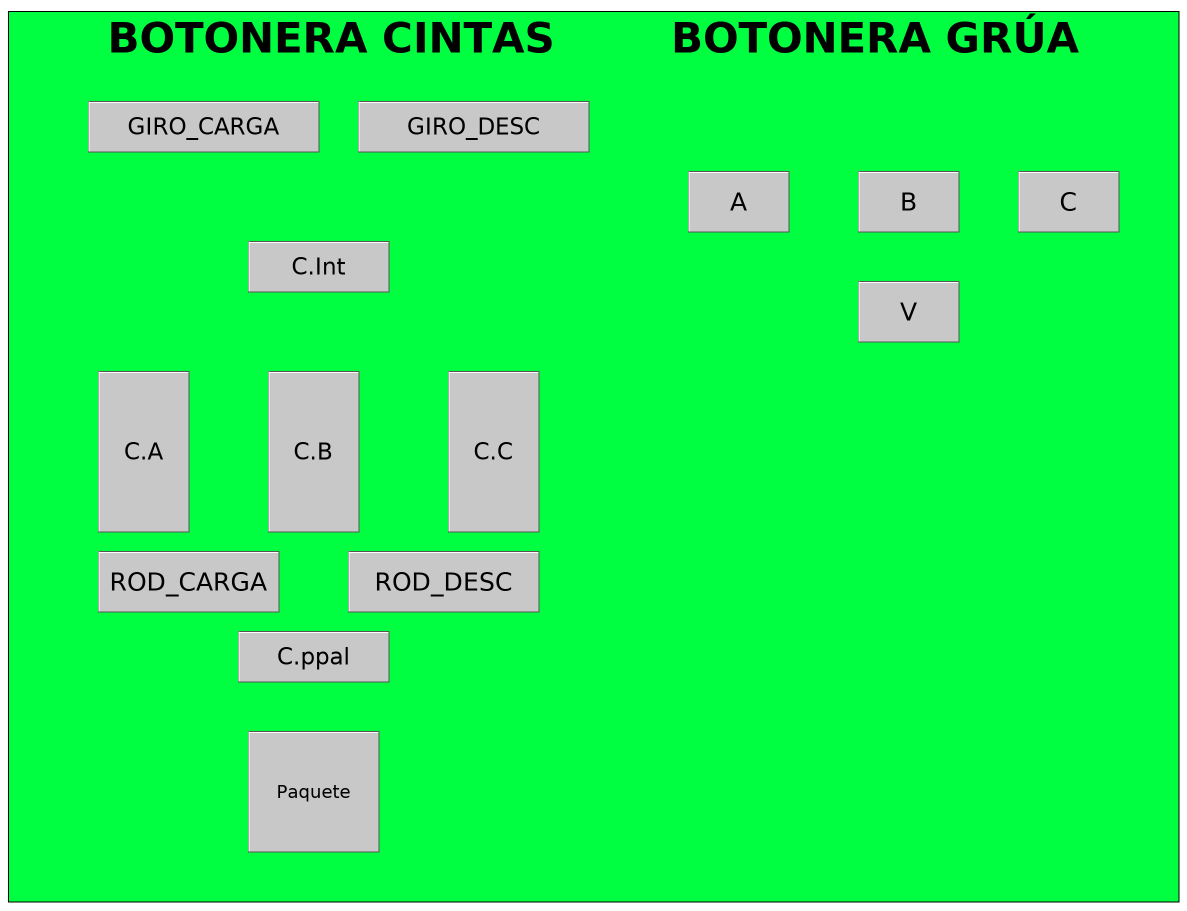
rectangle at (180,290)-(1351,1181): text "BOTONERA CINTAS        BOTONERA GRÚA"
button at (420,1010)-(551,1131): text "Paquete"; taps b_paquete
button at (410,910)-(561,961): text "C.ppal"; toggles b_acp
button at (270,650)-(361,811): text "C.A"; toggles b_aca
button at (620,650)-(711,811): text "C.C"; toggles b_acc
button at (420,520)-(561,571): text "C.Int"; toggles b_acint
button at (440,650)-(531,811): text "C.B"; toggles b_acb
button at (860,450)-(961,511): text "A"; taps b_B21
button at (1030,450)-(1131,511): text "B"; taps b_B22
button at (1190,450)-(1291,511): text "C"; taps b_B23
button at (1030,560)-(1131,621): text "V"; taps b_B24
button at (260,380)-(491,431): text "GIRO_CARGA"; toggles b_GirarIZQ
button at (530,380)-(761,431): text "GIRO_DESC"; toggles b_Volver1
button at (270,830)-(451,891): text "ROD_CARGA"; toggles b_rod_carga
button at (520,830)-(711,891): text "ROD_DESC"; toggles b_rod_desc
*)

(* Visualisation Botonera_pedidos
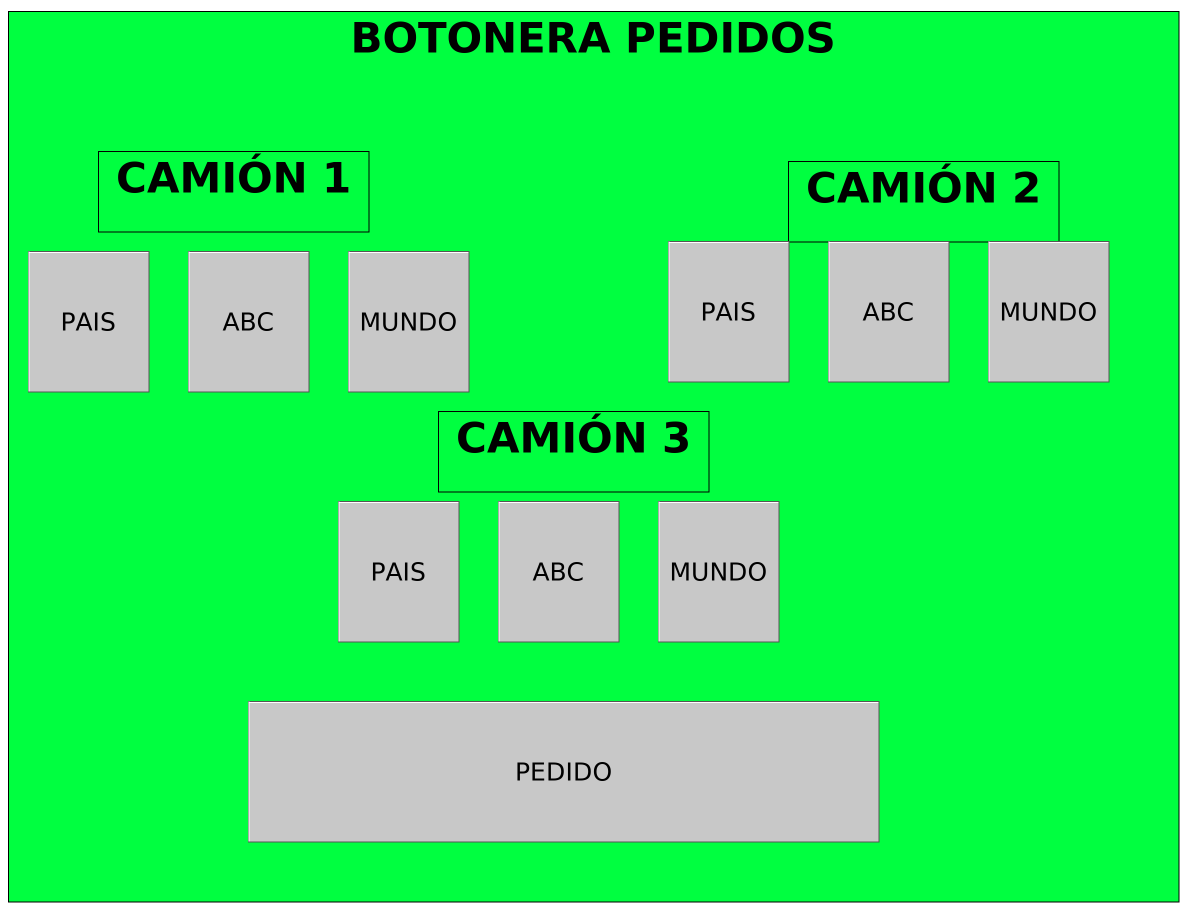
rectangle at (20,130)-(1191,1021): text "BOTONERA PEDIDOS"
button at (200,370)-(321,511): text "ABC"; taps b_c1abc
button at (360,370)-(481,511): text "MUNDO"; taps c1_mundo
button at (40,370)-(161,511): text "PAIS"; taps b_c1pais
button at (260,820)-(891,961): text "PEDIDO"; toggles pedido
rectangle at (110,270)-(381,351): text "CAMIÓN 1"
rectangle at (800,280)-(1071,361): text "CAMIÓN 2"
rectangle at (450,530)-(721,611): text "CAMIÓN 3"
button at (840,360)-(961,501): text "ABC"; taps b_c2abc
button at (510,620)-(631,761): text "ABC"; taps b_c3abc
button at (670,620)-(791,761): text "MUNDO"; taps b_c3mundo
button at (1000,360)-(1121,501): text "MUNDO"; taps b_c2mundo
button at (350,620)-(471,761): text "PAIS"; taps b_c3pais
button at (680,360)-(801,501): text "PAIS"; taps b_c2pais
*)

(* Visualisation ModosFunc
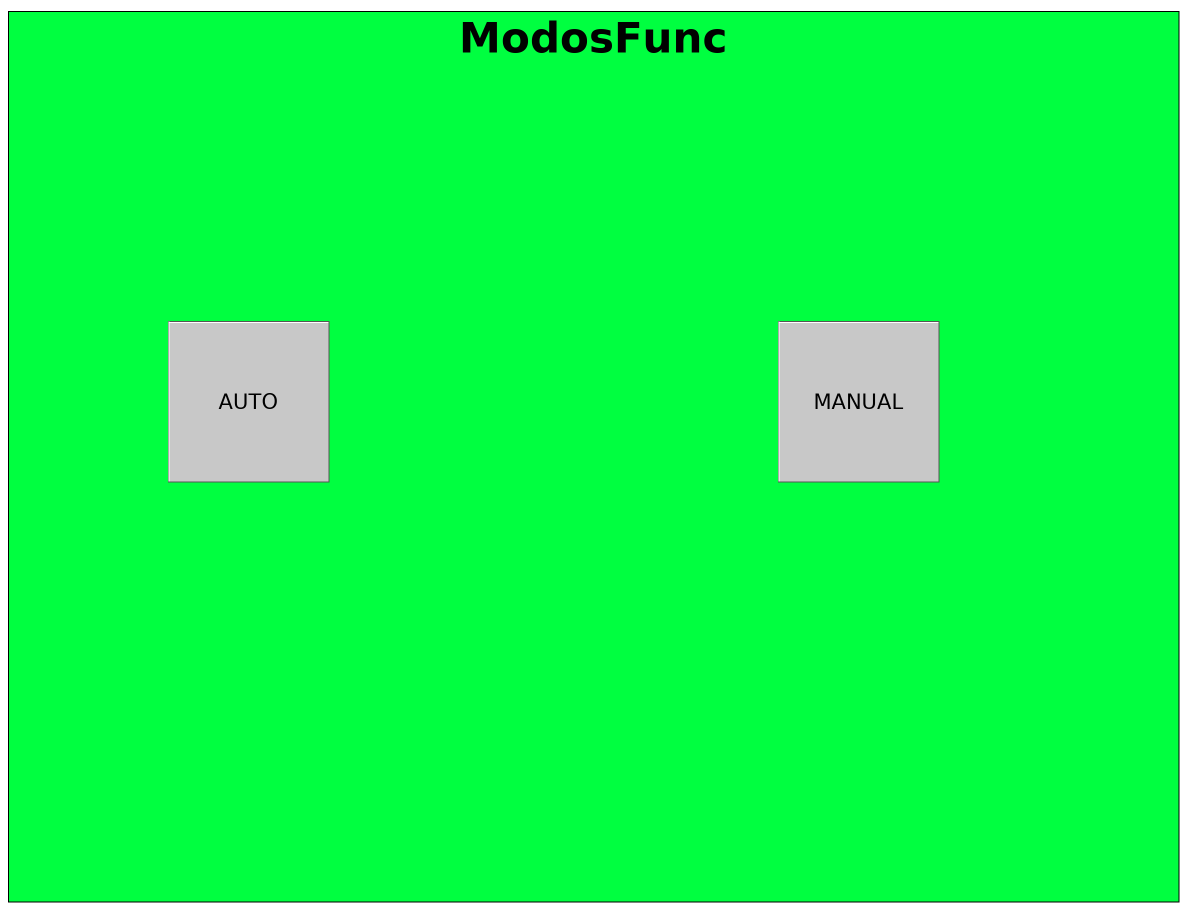
rectangle at (320,190)-(1491,1081): text "ModosFunc"
button at (480,500)-(641,661): text "AUTO"; toggles b_manual
button at (1090,500)-(1251,661): text "MANUAL"; toggles b_automatico
*)
